(* CODESYS project CodesysV3.export

Project tree, tasks and I/O mapping:
  application HomeAutomation
    libraries: Standard, * (System); Element Collections, 3.5.14.0 (3S - Smart Software Solutions GmbH); WagoSysStandard, 1.6.1.0 (WAGO); WagoTypesAppLED, 1.5.2.0 (WAGO); WagoAppAppLED, 1.7.2.0 (WAGO); WagoAppPlcModbus, 1.1.2.5 (WAGO); Util, 3.5.14.0 (System); BASIC, 3.3.4.0 (OSCAT); BUILDING, 1.0.0.1 (OSCAT); Common Helper for development, 1.1.0.5 (Stefan Dreyer); NETWORK, 1.3.5.3 (OSCAT); MQTT, 1.2.0.6 (Stefan Dreyer); WagoTypesEvent, 1.5.2.0 (WAGO); SysSocketAsync, 3.5.17.0 (System); SysTarget, 3.5.17.0 (System); SysSocket, * (System); SM3_Shared, 4.9.0.0 (3S - Smart Software Solutions GmbH); PRO JSON, 1.0.0.15 (Pro Electric)
    task MainTask (cyclic, interval 50 ms, priority 4) calls PLC_PRG_MAIN
    task MqttCommunication (freewheeling, priority 5) calls PLC_PRG_MQTT, DMX_SEND
    task Ping (cyclic, interval 10000 ms, priority 4) calls PRG_PING_DMX
    task RS485 (cyclic, interval 200 ms, priority 15) calls PLC_PRG_RS485
    PRG's/
      program DMX_SEND [ST]
      program PLC_PRG_MAIN [SFC]: MAIN_INIT, MOVE_COVERS, PROCESS_VIRTUAL, READ_PUSHBUTTONS, WRITE_SWITCHES
      program PLC_PRG_MQTT [SFC]: MQTT_INIT, MQTT_PUBLISH, MQTT_SUBSCRIBE
      program PLC_PRG_RS485 [SFC]: RS485_INIT, RS485_RUN
      program PRG_PING_DMX [ST]
    global variables DMXVariables
    global variables MqttVariables
    global variables PersistentVars
  data type Dimmer
  data type DIMMER_CURVE
  data type VIRTUAL_MODES
  Mqtt/
    data type MQTT_MESSAGE
    function block FB_MqttPublishQueue [ST]: AddMessage, GetMessage, Reset
    function block FB_MqttPublishWorker [ST]: Init, PublishMessage
  MqttDiscovery/
    Messages/
      data type MQTT_DISCOVERY_AVTY_T
      data type MQTT_DISCOVERY_BASE
      data type MQTT_DISCOVERY_BINARY_SENSOR
      data type MQTT_DISCOVERY_BINARY_SENSOR_ENT_CAT
      data type MQTT_DISCOVERY_COVER
      data type MQTT_DISCOVERY_DEVICE
      data type MQTT_DISCOVERY_LIGHT
      data type MQTT_DISCOVERY_LIGHT_DIMMER
      data type MQTT_DISCOVERY_LOCK
      data type MQTT_DISCOVERY_SENSOR
      data type MQTT_DISCOVERY_SENSOR_ENT_CAT
      data type MQTT_DISCOVERY_SIREN
      data type MQTT_DISCOVERY_SWITCH
  RS485/
    data type RS485_EASTRON_SDM_Devices
    data type RS485_RtuQuery
    interface RS485Device: GetRtuQuery, ProcessDataArray, RequestBusTime
    function block FB_RS485_BUSCONTROLLER [ST]: Init, RegisterDevice, ReleaseBus, SetBusOccupied
  function block FB_BASE_MQTT_DISCOVERY_DEVICE [ST]: CreateBinarySensorEntity, CreateBinarySensorEntityWithCategory, CreateCoverEntity, CreateLightDimmerEntity, CreateLightEntity, CreateLockEntity, CreateSensorEntity, CreateSensorEntityWithCategory, CreateSirenEntity, CreateSwitchEntity, initBaseDevice, SendLogMessage
  function block FB_INPUT_BINARYSENSOR_MQTT [ST]: ConfigureFunctionBlock, InitMqtt, InitMqttDiscovery
  function block FB_INPUT_PUSHBUTTON_DIMMER_MQTT [ST]: ConfigureFunctionBlock, InitMqtt
  function block FB_INPUT_PUSHBUTTON_MQTT [ST]: ConfigureFunctionBlock, InitMqtt, InitMqttDiscovery
  function block FB_MQTT_BASE [ST]: InitBaseMqtt
  function block FB_MQTT_LOG [ST]: InitMqtt, InitMqttDiscovery, send
  function block FB_OUTPUT_BINARY_MQTT [ST]: InitMqtt, InitMqttDiscoveryAsLight, InitMqttDiscoveryAsLock, InitMqttDiscoveryAsSiren, InitMqttDiscoveryAsSwitch, PublishReceived
  function block FB_OUTPUT_BISTABLE_MQTT [ST]: ConfigureFunctionBlock, InitMqtt, InitMqttDiscoveryAsLight, InitMqttDiscoveryAsLock, InitMqttDiscoveryAsSiren, InitMqttDiscoveryAsSwitch, PublishReceived
  function block FB_OUTPUT_COVER_MQTT [ST]: ConfigureFunctionBlock, InitMqtt, InitMqttDiscovery, PublishReceived
  function block FB_OUTPUT_DIMMER_MQTT [ST]: ConfigureFunctionBlock, initDMX, InitMqtt, InitMqttDiscovery, PublishReceived
  function block FB_PLC_MQTT_DISCOVERY_DEVICE [ST]: GetIpAddress, GetMac, initPlcDevice
  function block FB_RS485_DUCO_DUCOBOX_MQTT [ST]: AddNode, GetRtuQuery, InitMqtt, InitRS485, ProcessDataArray, PublishReceived, PubMqttMessage, RequestBusTime
  function block FB_RS485_DUCO_DUCOBOX_NODE_MQTT [ST]: GetRtuQuery, InitMqtt, InitNode, ProcessDataArray, PubMqttMessage, RequestBusTime
  function block FB_RS485_EASTRON_SDM_POWER_MQTT [ST]: GetRtuQuery, InitMqtt, InitRS485, ProcessDataArray, PubMqttMessage, RequestBusTime
  function block FB_RS485_EASTRON_SDM220_MQTT [ST]: GetRtuQuery, InitMqtt, InitRS485, ProcessDataArray, PubMqttMessage, RequestBusTime
  function block FB_RS485_ESERA_1WIRE_GATEWAY_MQTT [ST]: EnableOwd, GetRtuQuery, InitMqtt, InitRS485, ProcessDataArray, RequestBusTime
  function block FB_RS485_ESERA_OWD_MQTT [ST]: GetRtuQuery, InitMqtt, InitOwd, ProcessAirQuality, ProcessBrigthness, ProcessDataArray, ProcessDewPoint, ProcessHumidity, ProcessOwdVoltage, ProcessTemperature, PubMqttMessage, RequestBusTime
  function block FB_VIRTUAL_BOOL_MQTT [ST]: ConfigureFunctionBlockAsVirtualInput, ConfigureFunctionBlockAsVirtualOutput, InitMqtt, PublishReceived, SetValue
  function block FB_VIRTUAL_INT_MQTT [ST]: ConfigureFunctionBlockAsVirtualInput, ConfigureFunctionBlockAsVirtualOutput, InitMqtt, PublishReceived, SetValue
  function block FB_VIRTUAL_REAL_MQTT [ST]: ConfigureFunctionBlockAsVirtualInput, ConfigureFunctionBlockAsVirtualOutput, InitMqtt, PublishReceived, SetValue
  function block FB_VIRTUAL_STRING_MQTT [ST]: ConfigureFunctionBlockAsVirtualInput, ConfigureFunctionBlockAsVirtualOutput, InitMqtt, PublishReceived, SetValue
  function SwapWordsToReal [ST]
*)

// Dimmer
{attribute 'to_string' := ''}
TYPE Dimmer :
(
	idle,
	soft_turn_on_restore,
	soft_turn_off,
	quick_turn_on,
	quick_turn_off,
	ramp_up_or_down,
	low_or_high_entering,
	low_or_high_leaving,
	low_or_high_released_by_user,
	blink
);
END_TYPE

// DIMMER_CURVE
TYPE DIMMER_CURVE :
(
	linear,
	logarithmic,
	cubic
);
END_TYPE

// VIRTUAL_MODES
TYPE VIRTUAL_MODES :
(
	Input,
	Output
);
END_TYPE

// Mqtt/MQTT_MESSAGE
TYPE MQTT_MESSAGE :
STRUCT
	Payload: STRING(1500);
	Topic: STRING(128);
	Qos: MQTT.QoS;
	MqttRetain: BOOL;
END_STRUCT
END_TYPE

// RS485/RS485_EASTRON_SDM_Devices
TYPE RS485_EASTRON_SDM_Devices :
(
	SDM120,
	SDM220,
	SDM630
);
END_TYPE

// RS485/RS485_RtuQuery
TYPE RS485_RtuQuery :
STRUCT
	DeviceId: BYTE;
	FunctionCode: BYTE;
	ReadAddress: UINT;
	ReadQuantity: UINT;
	WriteAddress: UINT;
	WriteQuantity: UINT;
	WriteData: ARRAY[0..124] OF WORD;
END_STRUCT
END_TYPE

// MqttDiscovery/Messages/MQTT_DISCOVERY_AVTY_T
TYPE MQTT_DISCOVERY_AVTY_T :
STRUCT
	topic: JSONVAR;
END_STRUCT
END_TYPE

// MqttDiscovery/Messages/MQTT_DISCOVERY_BASE
TYPE MQTT_DISCOVERY_BASE :
STRUCT
	name: JSONVAR;
	/// object_id
	obj_id: JSONVAR;
	///unique_id
	uniq_id: JSONVAR;
	/// availability
	avty: ARRAY[1..2] OF MQTT_DISCOVERY_AVTY_T;
	/// availability mode
	avty_mode: JSONVAR;
	///payload_available
	pl_avail: JSONVAR;
	/// payload_not_available
	pl_not_avail: JSONVAR;
	/// device
	dev: MQTT_DISCOVERY_DEVICE;
	/// mqtt qos
	qos: JSONVAR;
	/// extra metadata
	meta: JSONVAR;
END_STRUCT
END_TYPE

// MqttDiscovery/Messages/MQTT_DISCOVERY_BINARY_SENSOR
TYPE MQTT_DISCOVERY_BINARY_SENSOR EXTENDS MQTT_DISCOVERY_BASE :
STRUCT
	///state_topic
	stat_t: JSONVAR;
	///payload_on
	pl_on: JSONVAR;
	///payload_off
	pl_off: JSONVAR;
	/// device class
	dev_cla: JSONVAR;
END_STRUCT
END_TYPE

// MqttDiscovery/Messages/MQTT_DISCOVERY_BINARY_SENSOR_ENT_CAT
TYPE MQTT_DISCOVERY_BINARY_SENSOR_ENT_CAT EXTENDS MQTT_DISCOVERY_BINARY_SENSOR :
STRUCT
	/// entity category
	ent_cat: JSONVAR;
END_STRUCT
END_TYPE

// MqttDiscovery/Messages/MQTT_DISCOVERY_COVER
TYPE MQTT_DISCOVERY_COVER EXTENDS MQTT_DISCOVERY_BASE :
STRUCT
	///command_topic
	cmd_t: JSONVAR;
	/// payload open
	pl_open: JSONVAR;
	/// payload_close
	pl_cls: JSONVAR;
	/// payload_stop
	pl_stop: JSONVAR;
	/// state topic
	stat_t: JSONVAR;
	/// state open
	stat_open: JSONVAR;
	/// state closed	
	stat_clsd: JSONVAR;
	///  optimistic
	opt: JSONVAR;
	/// device class
	dev_cla: JSONVAR;
END_STRUCT
END_TYPE

// MqttDiscovery/Messages/MQTT_DISCOVERY_DEVICE
TYPE MQTT_DISCOVERY_DEVICE :
STRUCT
	name: JSONVAR;
	///configuration_url
	cu: JSONVAR;
	///identifiers
	ids: JSONVAR;
	///manufacturer
	mf: JSONVAR;
	///model
	mdl: JSONVAR;
	///sw_version
	sw: JSONVAR;
	///hw_version
	hw: JSONVAR;
END_STRUCT
END_TYPE

// MqttDiscovery/Messages/MQTT_DISCOVERY_LIGHT
TYPE MQTT_DISCOVERY_LIGHT EXTENDS MQTT_DISCOVERY_BASE :
STRUCT
	///command_topic
	cmd_t: JSONVAR;
	/// payload_on
	pl_on: JSONVAR;
	/// payload_off
	pl_off: JSONVAR;
	/// state_topic
	stat_t: JSONVAR;
	///  optimistic
	opt: JSONVAR;
END_STRUCT
END_TYPE

// MqttDiscovery/Messages/MQTT_DISCOVERY_LIGHT_DIMMER
TYPE MQTT_DISCOVERY_LIGHT_DIMMER EXTENDS MQTT_DISCOVERY_LIGHT :
STRUCT
	///brightness state topic
	bri_stat_t: JSONVAR;
	/// brightness command topic
	bri_cmd_t: JSONVAR;
	/// brightness scale
	bri_scl: JSONVAR;
	/// on command type
	on_cmd_type: JSONVAR;
	/// DMX
	dmxChannel: JSONVAR;
	dmxWidth: JSONVAR;
	dmxUniverse: JSONVAR;
END_STRUCT
END_TYPE

// MqttDiscovery/Messages/MQTT_DISCOVERY_LOCK
TYPE MQTT_DISCOVERY_LOCK EXTENDS MQTT_DISCOVERY_BASE :
STRUCT
	///command_topic
	cmd_t: JSONVAR;
	/// payload lock
	pl_lock: JSONVAR;
	/// payload unlock
	pl_unlk: JSONVAR;
	/// state_topic
	stat_t: JSONVAR;
	/// state locked
	stat_locked: JSONVAR;
	/// state unlocked
	stat_unlocked: JSONVAR;
	///  optimistic
	opt: JSONVAR;
END_STRUCT
END_TYPE

// MqttDiscovery/Messages/MQTT_DISCOVERY_SENSOR
TYPE MQTT_DISCOVERY_SENSOR EXTENDS MQTT_DISCOVERY_BASE :
STRUCT
	///state_topic
	stat_t: JSONVAR;
	///expire after
	exp_aft: JSONVAR;
END_STRUCT
END_TYPE

// MqttDiscovery/Messages/MQTT_DISCOVERY_SENSOR_ENT_CAT
TYPE MQTT_DISCOVERY_SENSOR_ENT_CAT EXTENDS MQTT_DISCOVERY_SENSOR :
STRUCT
	/// entity category
	ent_cat: JSONVAR;
END_STRUCT
END_TYPE

// MqttDiscovery/Messages/MQTT_DISCOVERY_SIREN
TYPE MQTT_DISCOVERY_SIREN EXTENDS MQTT_DISCOVERY_BASE :
STRUCT
	///command_topic
	cmd_t: JSONVAR;
	/// payload_on
	pl_on: JSONVAR;
	/// payload_off
	pl_off: JSONVAR;
	/// state_topic
	stat_t: JSONVAR;
	/// state on
	stat_on: JSONVAR;
	/// state off
	stat_off: JSONVAR;
	///  optimistic
	opt: JSONVAR;
END_STRUCT
END_TYPE

// MqttDiscovery/Messages/MQTT_DISCOVERY_SWITCH
TYPE MQTT_DISCOVERY_SWITCH EXTENDS MQTT_DISCOVERY_BASE :
STRUCT
	///command_topic
	cmd_t: JSONVAR;
	/// payload_on
	pl_on: JSONVAR;
	/// payload_off
	pl_off: JSONVAR;
	/// state_topic
	stat_t: JSONVAR;
	/// state on
	stat_on: JSONVAR;
	/// state off
	stat_off: JSONVAR;
	///  optimistic
	opt: JSONVAR;
	/// device class
	dev_cla: JSONVAR;
END_STRUCT
END_TYPE

// HomeAutomation/DMXVariables
{attribute 'qualified_only'}
VAR_GLOBAL
	// unicast: 10.1.1.4
	// multicast: 10.1.1.255  
	// broadcast: 255.255.255.255  
	IP						: STRING:='10.1.1.4'; 
	DMX 					: oscat_network.NETWORK_BUFFER_SHORT;
END_VAR

// HomeAutomation/MqttVariables
{attribute 'qualified_only'}
VAR_GLOBAL	
	(* Broker setup *)
	clientID				:STRING:='PLC-House';
	broker					:STRING:='192.168.1.52:1883'; 	
	(* use the below for username password authentication to broker *)
	(* broker					:STRING:='user:password@192.168.1.36:1883'; *)
	

	(* Shared Variables for MQTT publish communication *)
	fbMqttPublishQueue		:FB_MqttPublishQueue;  
	
	(* Shared Variables for MQTT subscribe communication *)	
	collector_FB_OUTPUT_SWITCH_MQTT		:MQTT.CallbackCollector;		
	collector_FB_OUTPUT_COVER_MQTT		:MQTT.CallbackCollector;	
	collector_FB_VIRTUAL_MQTT			:MQTT.CallbackCollector;		
	collector_FB_DIMMER_MQTT			:MQTT.CallbackCollector;
	collector_FB_MQTT_LOG				:MQTT.CallbackCollector;	
	collector_FB_RS485_MQTT				:MQTT.CallbackCollector;
	
	(* QOS Constants *)
	MQTT_QOS_EXACTLY_ONCE				:MQTT.QoS := MQTT.QoS.ExactlyOnce;
	 
	
	(* HOME ASSISTANT DISCOVERY VIA MQTT*)
	PLC_Device						:FB_PLC_MQTT_DISCOVERY_DEVICE;	
	
	(* Topics *)
	MqttMain						:STRING(16) := 'Devices/';
	MqttType						:STRING(16) := 'PLC/';
	MqttDevice						:STRING(16) := 'House/';
	// e.g. Devices/PLC/House
	MqttBaseTopic					:STRING(100) := CONCAT(CONCAT(MqttMain,MqttType),MqttDevice);
	MqttDiagnosticTopic				:STRING(100) := CONCAT(MqttBaseTopic,'diagnostic');									
	MqttAvailabilityTopic 			:STRING(100) := CONCAT(MqttBaseTopic,'availability');							
	MqttAvailabilityOnlinePayload	:STRING(20) := 'online';							
	MqttAvailabilityOfflinePayload	:STRING(20) := 'offline';
	MQTTAvailabilityHartbeatTime	:TIME:=T#5S;
	MqttHADiscoveryPrefix			:STRING(16) := 'homeassistant/';
	
	(* FB Topics *)
	MqttPushbuttonPrefix			:STRING(100) := CONCAT(MqttBaseTopic,'Out/DigitalInputs/Pushbuttons/');
	MqttPubSwitchPrefix				:STRING(100) := CONCAT(MqttBaseTopic,'Out/DigitalOutputs/');
	MqttSubSwitchPrefix				:STRING(100) := CONCAT(MqttBaseTopic,'In/DigitalOutputs/');
	MqttPubCoverPrefix				:STRING(100) := CONCAT(MqttBaseTopic,'Out/Covers/');
	MqttSubCoverPrefix				:STRING(100) := CONCAT(MqttBaseTopic,'In/Covers/');
	MqttPubDimmerPrefix				:STRING(100) := CONCAT(MqttBaseTopic,'Out/Dimmers/');
	MqttSubDimmerPrefix				:STRING(100) := CONCAT(MqttBaseTopic,'In/Dimmers/');
	MqttPubVirtualPrefix			:STRING(100) := CONCAT(MqttBaseTopic,'Out/Virtuals/');
	MqttSubVirtualPrefix			:STRING(100) := CONCAT(MqttBaseTopic,'In/Virtuals/');
	MqttPubRS485Prefix				:STRING(100) := CONCAT(MqttBaseTopic,'Out/RS485/');
	MqttSubRS485Prefix				:STRING(100) := CONCAT(MqttBaseTopic,'In/RS485/');
	
	(* Wildcard subscriptions *)
	MqttSubSwitchTopic				:STRING(100) := CONCAT(MqttSubSwitchPrefix,'+');
	MqttSubCoverTopic				:STRING(100) := CONCAT(MqttSubCoverPrefix,'+');
	MqttSubVirtualTopic				:STRING(100) := CONCAT(MqttSubVirtualPrefix,'+');
	MqttSubDimmerTopic				:STRING(100) := CONCAT(MqttSubDimmerPrefix,'#');
	MqttSubRS485Topic				:STRING(100) := CONCAT(MqttSubRS485Prefix,'#');

END_VAR

// HomeAutomation/PersistentVars
{attribute 'qualified_only'}
VAR_GLOBAL PERSISTENT RETAIN
	// Generated instance path of persistent variable
	PLC_PRG_MAIN.FB_DO_BIN_001.PreviousState: BOOL;
	// Generated instance path of persistent variable
	PLC_PRG_MAIN.FB_DO_COVER_001.internalDir: BOOL;
	// Generated instance path of persistent variable
	PLC_PRG_MAIN.FB_AO_DIMMER_001.PreviousOUT: BYTE;
	// Generated instance path of persistent variable
	PLC_PRG_MAIN.FB_AO_DIMMER_001.PreviousQ: BOOL;
	// Generated instance path of persistent variable
	PLC_PRG_MAIN.FB_VIRTUAL_INT_001.PreviousState: INT;
	// Generated instance path of persistent variable
	PLC_PRG_MAIN.FB_VIRTUAL_BOOL_001.PreviousState: BOOL;
	// Generated instance path of persistent variable
	PLC_PRG_MAIN.FB_VIRTUAL_STRING_001.PreviousState: STRING;
	// Generated instance path of persistent variable
	PLC_PRG_MAIN.FB_VIRTUAL_REAL_001.PreviousState: REAL;
END_VAR

// HomeAutomation/PRG's/PLC_PRG_MAIN
PROGRAM PLC_PRG_MAIN
VAR		
	(* INPUT FUNCTION BLOCKS *)
	FB_DI_PB_001				:FB_INPUT_PUSHBUTTON_MQTT;
	FB_DI_PB_002				:FB_INPUT_PUSHBUTTON_DIMMER_MQTT;
	
	(* OUTPUT FUNCTION BLOCKS *)
	FB_DO_BIN_001				:FB_OUTPUT_BINARY_MQTT;
	FB_DO_BISTABLE_001			:FB_OUTPUT_BISTABLE_MQTT;

	(* COVER FUNCTION BLOCKS *)
	FB_DO_COVER_001				:FB_OUTPUT_COVER_MQTT;
	
	(* DIMMER FUNCTION BLOCKS *)
	FB_AO_DIMMER_001			:FB_OUTPUT_DIMMER_MQTT;	
	TestOUT						:WORD;
	
	(* VIRTUAL FUNCTION BLOCKS *)
	FB_VIRTUAL_INT_001				:FB_VIRTUAL_INT_MQTT;
	FB_VIRTUAL_BOOL_001				:FB_VIRTUAL_BOOL_MQTT;
	FB_VIRTUAL_STRING_001			:FB_VIRTUAL_STRING_MQTT;
	FB_VIRTUAL_REAL_001				:FB_VIRTUAL_REAL_MQTT;
END_VAR

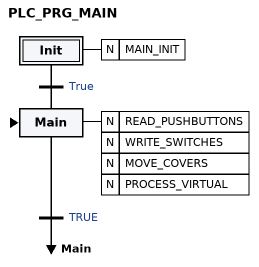
INITIAL_STEP Init:
    MAIN_INIT(N);
END_STEP
TRANSITION FROM Init TO Main
    := True;
END_TRANSITION
STEP Main:
    READ_PUSHBUTTONS(N);
    WRITE_SWITCHES(N);
    MOVE_COVERS(N);
    PROCESS_VIRTUAL(N);
END_STEP
TRANSITION FROM Main TO Main
    := TRUE;
END_TRANSITION

ACTION MAIN_INIT:
(* MQTT Discovery device*)
MqttVariables.PLC_Device.initPlcDevice(
	MqttDiscoveryPrefix := MqttVariables.MqttHADiscoveryPrefix,
	pMqttPublishQueue := ADR(MqttVariables.fbMqttPublishQueue),
	availabilityTopic := MqttVariables.MqttAvailabilityTopic,
	availabilityOnline := MqttVariables.MqttAvailabilityOnlinePayload,
	availabilityOffline := MqttVariables.MqttAvailabilityOfflinePayload,
	MqttDiagnosticTopic := MqttVariables.MqttDiagnosticTopic
);


(* INIT DIGITAL INPUT STUFF *)
FB_DI_PB_001.InitMqtt(
	MQTTPublishPrefix:= ADR(MqttVariables.MqttPushbuttonPrefix),	(* pointer to string prefix for the mqtt publish topic *)
	pMqttPublishQueue := ADR(MqttVariables.fbMqttPublishQueue)		(* pointer to MqttPublishQueue to send a new Mqtt event *)
);

FB_DI_PB_001.InitMqttDiscovery(
	name := 'Button number 001',						(* The name show in Home Assistant frond-end*)
	Device := ADR(MqttVariables.PLC_Device),							(* The device show in Home Assistant *)
);

FB_DI_PB_002.InitMqtt(
	MQTTPublishPrefix:= ADR(MqttVariables.MqttPushbuttonPrefix),	
	pMqttPublishQueue := ADR(MqttVariables.fbMqttPublishQueue),
    TRUE,                                                               (* specify whether dimmer value should be outputted on MQTT topic *)
    MQTT.QoS.ExactlyOnce,                                            (* specify the QoS for the dimmer mqtt events (values 0-255) *)    
    5                                                                   (* specify the resolution for the dimmer mqtt events *)    
);


(* ALTER THE DIMMER OUTPUT DEFAULT BEHAVIOR *)
FB_AO_DIMMER_001.ConfigureFunctionBlock(
	T_Debounce:=T#10MS,
	T_Reconfig:=T#10S,
	T_On_Max:=T#0S,
	T_Dimm_Start:=T#400MS,
	T_Dimm:=T#3S,
	Min_On:=50,
	Max_On:=255,
	Soft_Dimm:=TRUE,
	Rst_Out:=FALSE,
	OUT_LinearScaleMin:=11000,
	OUT_LinearScaleMax:=32767
);

(* INIT DMX / ART-NET OUTPUT, OPTIONAL*)
FB_AO_DIMMER_001.InitDmx(
	DmxChannel := 1,							(* The channel *)
	DmxWidth:=1, 								(* Width of DMX channel, 1 or 2, aka 8 or 16 bit *)
	pDmxValues := ADR(DMXVariables.DMX.BUFFER), (* pointer to network buffer *)
	DmxUniverse:=1								(* Universe, but the buffer desides, this is only meta data that ends up in MQTT*)
);

(* INIT HOME ASSISTANT DISCOVERTY*)
FB_AO_DIMMER_001.InitMqttDiscovery(
	name := '001. Office strip cold',					(* The name show in Home Assistant frond-end*)
	Device := ADR(MqttVariables.PLC_Device),							(* The device show in Home Assistant *)
);


(* INIT DIGITAL OUTPUT STUFF *)
FB_DO_BISTABLE_001.InitMqtt(
	MQTTPublishPrefix:= ADR(MqttVariables.MqttPubSwitchPrefix),					(* pointer to string prefix for the mqtt publish topic *)
	MQTTSubscribePrefix:= ADR(MqttVariables.MqttSubSwitchPrefix),				(* pointer to string prefix for the mqtt subscribe topic *)
	pMqttPublishQueue := ADR(MqttVariables.fbMqttPublishQueue),					(* pointer to MqttPublishQueue to send a new Mqtt event *)
	pMqttCallbackCollector := ADR(MqttVariables.collector_FB_OUTPUT_SWITCH_MQTT)(* pointer to CallbackCollector to receive Mqtt subscription events *)
);

FB_DO_BISTABLE_001.InitMqttDiscoveryAsLight(
	name := 'light number 1',						(* The name show in Home Assistant frond-end*)
	Device := ADR(MqttVariables.PLC_Device),							(* The device show in Home Assistant *)
);

FB_DO_BIN_001.InitMqtt(
	MQTTPublishPrefix:= ADR(MqttVariables.MqttPubSwitchPrefix),					(* pointer to string prefix for the mqtt publish topic *)
	MQTTSubscribePrefix:= ADR(MqttVariables.MqttSubSwitchPrefix),				(* pointer to string prefix for the mqtt subscribe topic *)
	pMqttPublishQueue := ADR(MqttVariables.fbMqttPublishQueue),					(* pointer to MqttPublishQueue to send a new Mqtt event *)
	pMqttCallbackCollector := ADR(MqttVariables.collector_FB_OUTPUT_SWITCH_MQTT)(* pointer to CallbackCollector to receive Mqtt subscription events *)
);

FB_DO_BIN_001.InitMqttDiscoveryAsLight(
	name := 'light number 2',						(* The name show in Home Assistant frond-end*)
	Device := ADR(MqttVariables.PLC_Device),							(* The device show in Home Assistant *)
);

(* INIT COVERS STUFF *)
FB_DO_COVER_001.InitMqtt(MQTTPublishPrefix:= ADR(MqttVariables.MqttPubCoverPrefix),	(* pointer to string prefix for the mqtt publish topic *)
	MQTTSubscribePrefix:= ADR(MqttVariables.MqttSubCoverPrefix),					(* pointer to string prefix for the mqtt subscribe topic *)
	pMqttPublishQueue := ADR(MqttVariables.fbMqttPublishQueue),						(* pointer to MqttPublishQueue to send a new Mqtt event *)
	pMqttCallbackCollector := ADR(MqttVariables.collector_FB_OUTPUT_COVER_MQTT)  	(* pointer to CallbackCollector to receive Mqtt subscription events *)
);

FB_DO_COVER_001.initmqttdiscovery(								(*see dimmer for full example *)
	name := 'cover number 001',									(* the name show in home assistant frond-end*)
	device := ADR(MqttVariables.PLC_Device),										(* the device show in home assistant *)
);

FB_DO_COVER_001.ConfigureFunctionBlock(
	T_LOCKOUT:=T#1S,											(* delay between change of direction *)
	T_UD:=T#20S													(* run time to move the cover completely up/down *)
);


(* INIT VIRTUAL STUFF *)
FB_VIRTUAL_STRING_001.InitMqtt(MQTTPublishPrefix:= ADR(MqttVariables.MqttPubVirtualPrefix),				
	MQTTSubscribePrefix:= ADR(MqttVariables.MqttSubVirtualPrefix),									
	pMqttPublishQueue := ADR(MqttVariables.fbMqttPublishQueue),						
	pMqttCallbackCollector := ADR(MqttVariables.collector_FB_VIRTUAL_MQTT),
	MqttQos:=MQTT.QoS.ExactlyOnce, 
	MqttRetain:=FALSE									
);
FB_VIRTUAL_STRING_001.ConfigureFunctionBlockAsVirtualInput(DefaultValue:='HelloWorld',SetDefaultValueStartup:=TRUE,PublishAtStartup:=TRUE,UsePersistentAtStartup:=FALSE,ConfirmReceival:=TRUE);


FB_VIRTUAL_INT_001.InitMqtt(MQTTPublishPrefix:= ADR(MqttVariables.MqttPubVirtualPrefix),				
	MQTTSubscribePrefix:= ADR(MqttVariables.MqttSubVirtualPrefix),									
	pMqttPublishQueue := ADR(MqttVariables.fbMqttPublishQueue),						
	pMqttCallbackCollector := ADR(MqttVariables.collector_FB_VIRTUAL_MQTT),
	MqttQos:=MQTT.QoS.ExactlyOnce, 
	MqttRetain:=FALSE												
);
FB_VIRTUAL_INT_001.ConfigureFunctionBlockAsVirtualInput(DefaultValue:=0,SetDefaultValueStartup:=TRUE,PublishAtStartup:=TRUE,UsePersistentAtStartup:=FALSE,ConfirmReceival:=TRUE);
(* FB_VIRTUAL_INT_001.ConfigureFunctionBlockAsVirtualOutput(PublishAtStartup:=TRUE); *)


FB_VIRTUAL_BOOL_001.InitMqtt(MQTTPublishPrefix:= ADR(MqttVariables.MqttPubVirtualPrefix),				
	MQTTSubscribePrefix:= ADR(MqttVariables.MqttSubVirtualPrefix),									
	pMqttPublishQueue := ADR(MqttVariables.fbMqttPublishQueue),						
	pMqttCallbackCollector := ADR(MqttVariables.collector_FB_VIRTUAL_MQTT),
	MqttQos:=MQTT.QoS.ExactlyOnce, 
	MqttRetain:=FALSE											
);
(* FB_VIRTUAL_BOOL_001.ConfigureFunctionBlockAsVirtualInput(DefaultValue:=FALSE,SetDefaultValueStartup:=TRUE,PublishAtStartup:=TRUE,UsePersistentAtStartup:=FALSE); *)
FB_VIRTUAL_BOOL_001.ConfigureFunctionBlockAsVirtualOutput(PublishAtStartup:=TRUE);

FB_VIRTUAL_REAL_001.InitMqtt(MQTTPublishPrefix:= ADR(MqttVariables.MqttPubVirtualPrefix),				
	MQTTSubscribePrefix:= ADR(MqttVariables.MqttSubVirtualPrefix),									
	pMqttPublishQueue := ADR(MqttVariables.fbMqttPublishQueue),						
	pMqttCallbackCollector := ADR(MqttVariables.collector_FB_VIRTUAL_MQTT),
	MqttQos:=MQTT.QoS.ExactlyOnce, 
	MqttRetain:=FALSE												
);
FB_VIRTUAL_REAL_001.ConfigureFunctionBlockAsVirtualInput(DefaultValue:=0.1,SetDefaultValueStartup:=TRUE,PublishAtStartup:=TRUE,UsePersistentAtStartup:=FALSE,ConfirmReceival:=TRUE);
(* FB_VIRTUAL_REAL_001.ConfigureFunctionBlockAsVirtualOutput(PublishAtStartup:=TRUE); *)



MqttVariables.PLC_Device.SendLogMessage('Init finished', 'MAIN_INIT');
END_ACTION

ACTION MOVE_COVERS:
FB_DO_COVER_001(
	TOGGLE:=FB_DI_PB_001.P_LONG,
	MU=>DO_031,
	MD=>DO_032	
);
END_ACTION

ACTION PROCESS_VIRTUAL:

FB_VIRTUAL_BOOL_001();
FB_VIRTUAL_INT_001();
FB_VIRTUAL_STRING_001();
FB_VIRTUAL_REAL_001();
END_ACTION

ACTION READ_PUSHBUTTONS:
FB_DI_PB_001(PB:= DI_001); (* Provide the input FB the correct phyical input to validate each cyclus *)
FB_DI_PB_002(PB:= DI_002);
END_ACTION

ACTION WRITE_SWITCHES:
FB_DO_BIN_001(OUT	=>		DO_001,										(* couple the function block to the physical output *)
	PRIO_HIGH				:=FALSE,  									(* brings the output high regardless of other input values *)
	PRIO_LOW				:=FALSE, 									(* brings the output low regardless of other input values. NOTE: PRIO_HIGH overrules PRIO_LOW input *)
	TOGGLE					:=FB_DI_PB_001.SINGLE 						(* for toggling the output *)	
);

FB_AO_DIMMER_001(
	SINGLE:=FB_DI_PB_001.SINGLE,
	LONG:=FB_DI_PB_001.LONG, 
	P_LONG:=FB_DI_PB_001.P_LONG, 
	Q_OUT => TestOUT,
	SET:=  FB_DI_PB_001.DOUBLE,
	VAL:=125
);

FB_DO_BISTABLE_001();
END_ACTION

END_PROGRAM

// FB_INPUT_PUSHBUTTON_MQTT
{attribute 'reflection' := ''}
FUNCTION_BLOCK FB_INPUT_PUSHBUTTON_MQTT EXTENDS FB_MQTT_BASE
VAR_INPUT
	PB: BOOL;
END_VAR
VAR_OUTPUT
	SINGLE: BOOL;
	DOUBLE: BOOL;
	LONG: BOOL;
	P_LONG: BOOL;
END_VAR
VAR
	/// Refelection: object's full instance name
	{attribute 'instance-path' := ''}
	{attribute 'noinit'}
	InstancePath: STRING;
	FB_DETECTPUSH: OSCAT_BUILDING.CLICK_MODE;
	P_LONG_R_TRIG: Standard.R_TRIG;
	P_LONG_F_TRIG: Standard.F_TRIG;
	/// Default value for click mode, can be overwritten by method call 
	T_Long: TIME := TIME#400ms;
	MqttDiscoveryMessage: MQTT_DISCOVERY_SENSOR;
END_VAR

FB_DETECTPUSH(
	IN:= PB, 	
	SINGLE=> SINGLE, 
	DOUBLE=> DOUBLE, 
	TP_LONG=> LONG, 
	LONG=> P_LONG,
	T_LONG:= T_Long);
	
P_LONG_R_TRIG(CLK:=FB_DETECTPUSH.LONG);
P_LONG_F_TRIG(CLK:=FB_DETECTPUSH.LONG);
	
IF FB_DETECTPUSH.SINGLE AND InitMqttDone THEN
	pMqttPublishQueue^.AddMessage(
		Payload := 'SINGLE',
		Topic := CONCAT(MqttPublishTopicPrefix^, MqttPublishTopicSuffix),
		Qos := MQTT.QoS.ExactlyOnce,
		MqttRetain := FALSE
	);
END_IF

IF FB_DETECTPUSH.DOUBLE AND InitMqttDone THEN
	pMqttPublishQueue^.AddMessage(
		Payload := 'DOUBLE',
		Topic := CONCAT(MqttPublishTopicPrefix^, MqttPublishTopicSuffix),
		Qos := MQTT.QoS.ExactlyOnce,
		MqttRetain := FALSE
	);
END_IF

IF FB_DETECTPUSH.TP_LONG AND InitMqttDone THEN
	pMqttPublishQueue^.AddMessage(
		Payload := 'LONG',
		Topic := MQTTPublishTopic,
		Qos := MQTT.QoS.ExactlyOnce,
		MqttRetain := FALSE
	);
END_IF

IF P_LONG_F_TRIG.Q AND InitMqttDone THEN
	pMqttPublishQueue^.AddMessage(
		Payload := 'RELEASED',
		Topic := MQTTPublishTopic,
		Qos := MQTT.QoS.ExactlyOnce,
		MqttRetain := FALSE
	);
END_IF



IF (P_LONG_R_TRIG.Q OR P_LONG_F_TRIG.Q) AND InitMqttDone THEN
	

	pMqttPublishQueue^.AddMessage(
		Payload := BOOL_TO_STRING(FB_DETECTPUSH.LONG),
		Topic := CONCAT(MQTTPublishTopic,'/P_LONG'),
		Qos := MQTT.QoS.ExactlyOnce,
		MqttRetain := TRUE
	);
END_IF

METHOD ConfigureFunctionBlock
VAR_INPUT
	/// Default value for click mode, can be overwritten by method call 
	T_Long: TIME;
END_VAR
THIS^.T_Long:=T_Long;
END_METHOD

METHOD InitMqtt
VAR_INPUT
	MQTTPublishPrefix: POINTER TO STRING;
	pMqttPublishQueue: POINTER TO FB_MqttPublishQueue;
END_VAR
SUPER^._InstancePath := THIS^.InstancePath; // Due to reflection its location is important

(*pass trough*)
THIS^.pMqttPublishQueue := pMqttPublishQueue;
THIS^.MqttPublishTopicPrefix:=MQTTPublishPrefix;
SUPER^.InitBaseMqtt();
END_METHOD

METHOD InitMqttDiscovery
VAR_INPUT
	Device: POINTER TO FB_PLC_MQTT_DISCOVERY_DEVICE;
	Name: STRING(255);
	overruleId: STRING(255) := '';
	meta: STRING(255) := '';
END_VAR
VAR
	id: STRING(255);
END_VAR
IF InitMqttDone AND NOT initMqttDiscoveryDone THEN
	
	IF CommonTypesAndFunctions.StrEquals(str1:= ADR(overruleId), str2:= ADR('')) THEN
		id := CONCAT(CONCAT(THIS^.DeviceName,'_'), THIS^.InstanceNamePt^); // 'FB_DI_PB_003'
	ELSE
		id := overruleId; // 'MY_PH_GND_HALL_01'
	END_IF
	
	Device^.CreateSensorEntity(
		Name := name,
		Id := id,
		Meta := meta,
		StateTopic := THIS^.MQTTPublishTopic,
		ExpiryAfter := 2);

	initMqttDiscoveryDone := TRUE;
END_IF
END_METHOD

END_FUNCTION_BLOCK

// FB_MQTT_BASE
FUNCTION_BLOCK FB_MQTT_BASE
VAR
	_InstancePath: STRING;
	InstanceNamePt: POINTER TO STRING;
	DeviceName: STRING;
	InitMqttDone: BOOL;
	/// Publish (Out);
	MqttPublishTopicPrefix: POINTER TO STRING;
	MqttPublishTopicSuffix: STRING(50);
	MQTTPublishTopic: STRING(100);
	/// Subscribe (In)
	MqttSubscribeTopicPrefix: POINTER TO STRING;
	MqttSubscribeTopicSuffix: STRING(50);
	MQTTSubscribeTopic: STRING(100);
	pMqttPublishQueue: POINTER TO FB_MqttPublishQueue;
	MqttHighRequest: BOOL;
	MqttLowRequest: BOOL;
	MqttQos: MQTT.QoS := MQTT.QoS.ExactlyOnce;
	MqttRetain: BOOL := TRUE;
	/// HA Discovery specific 
	ComposeJSON: STRUCT_TO_JSON;
	initMqttDiscoveryDone: BOOL := FALSE;
END_VAR

METHOD InitBaseMqtt
VAR
	MQTTPublishPrefix: POINTER TO STRING;
	MQTTSubscribePrefix: POINTER TO STRING;
	pMqttPublishQueue: POINTER TO FB_MqttPublishQueue;
END_VAR

(*Define instance names*)
InstanceNamePt := CommonTypesAndFunctions.FindLastDot(ADR(_InstancePath)) + 1;

DeviceName := LEFT(_InstancePath,find(_InstancePath, '.' )-1  ) ;

// Publish (Out);
IF	NOT CommonTypesAndFunctions.StrEquals(ADR(MqttPublishTopicPrefix),ADR('')) THEN
	THIS^.MqttPublishTopicSuffix := InstanceNamePt^;
	THIS^.MQTTPublishTopic := CONCAT(MqttPublishTopicPrefix^, THIS^.MqttPublishTopicSuffix);
END_IF

// Subscribe (In)
IF	NOT CommonTypesAndFunctions.StrEquals(ADR(MqttSubscribeTopicPrefix),ADR('')) THEN
	THIS^.MQTTSubscribeTopicSuffix := InstanceNamePt^;
	THIS^.MQTTSubscribeTopic := CONCAT(MqttSubscribeTopicPrefix^ ,THIS^.MQTTSubscribeTopicSuffix);
END_IF

InitMqttDone := TRUE;
END_METHOD

END_FUNCTION_BLOCK

// Mqtt/FB_MqttPublishQueue
FUNCTION_BLOCK FB_MqttPublishQueue
VAR_OUTPUT
	EMPTY: BOOL := TRUE;
	FULL: BOOL;
END_VAR
VAR
	localMessage: MQTT_MESSAGE;
	fifo: ARRAY[0..n] OF MQTT_MESSAGE;
	pr: INT;
	pw: INT;
END_VAR
VAR CONSTANT
	/// changing this value will chage the number of stored elements in the fifo 
	n: INT := 1024;
END_VAR

METHOD AddMessage
VAR_INPUT
	Payload: STRING(1500);
	Topic: STRING(128);
	Qos: MQTT.QoS;
	MqttRetain: BOOL;
END_VAR
IF NOT FULL THEN
	localMessage.Payload := Payload;
	localMessage.Topic := Topic;
	localMessage.Qos := Qos;
	localMessage.MqttRetain := MqttRetain;
	fifo[pw] := localMessage;
	pw := OSCAT_BASIC.INC1(pw,n);
	FULL := pw = pr;
	EMPTY := FALSE;
END_IF;
END_METHOD

METHOD GetMessage : MQTT_MESSAGE
IF NOT EMPTY THEN
	GetMessage := fifo[pr];
	pr := OSCAT_BASIC.INC1(pr,n);
	EMPTY := pr = pw;
	FULL := FALSE;
END_IF;
END_METHOD

METHOD Reset
pw := pr;
FULL := FALSE;
EMPTY := TRUE;
END_METHOD

END_FUNCTION_BLOCK

// FB_PLC_MQTT_DISCOVERY_DEVICE
{attribute 'reflection' := ''}
FUNCTION_BLOCK FB_PLC_MQTT_DISCOVERY_DEVICE EXTENDS FB_BASE_MQTT_DISCOVERY_DEVICE
VAR
	MqttDiagnosticTopicIP: STRING;
	MqttRefreshIP: OSCAT_BASIC.GEN_PULSE;
END_VAR

(* allow the pulse generator to generate a pulse, used for refreshing IP address *)
MqttRefreshIP();

(* Refresh the IP address on every pulse *)
IF NOT(xInit) AND MqttRefreshIP.Q THEN		
	pMqttPublishQueue^.AddMessage(
		Payload:= GetIpAddress(),
		Topic := MqttDiagnosticTopicIP,
		Qos := MQTT.QoS.ExactlyOnce,
		MqttRetain := TRUE,
	);
END_IF

METHOD PRIVATE GetIpAddress : STRING(15)
VAR
	AdapterInfo: SOCK_ADAPTER_INFORMATION;
	hAdapter: RTS_IEC_HANDLE;
	udiStructSize: UDINT := SIZEOF(AdapterInfo);
	rResult: RTS_IEC_RESULT;
	xFirstAdapter: BOOL;
END_VAR
xFirstAdapter := TRUE;
rResult := 0;
WHILE rResult = 0 DO   
	IF xFirstAdapter THEN
		hAdapter := SysSockGetFirstAdapterInfo(ADR(AdapterInfo), ADR(udiStructSize), ADR(rResult));
	ELSE   
		hAdapter := SysSockGetNextAdapterInfo(hAdapter, ADR(AdapterInfo), ADR(udiStructSize), ADR(rResult));
	END_IF
	IF rResult = 0 THEN
		GetIpAddress := Standard.CONCAT(BYTE_TO_STRING(AdapterInfo.IpAddr.S_un_b.s_b1),'.');
		GetIpAddress := Standard.CONCAT(GetIpAddress,BYTE_TO_STRING(AdapterInfo.IpAddr.S_un_b.s_b2));
		GetIpAddress := Standard.CONCAT(GetIpAddress,'.');
		GetIpAddress := Standard.CONCAT(GetIpAddress,BYTE_TO_STRING(AdapterInfo.IpAddr.S_un_b.s_b3));
		GetIpAddress := Standard.CONCAT(GetIpAddress,'.');
		GetIpAddress := Standard.CONCAT(GetIpAddress,BYTE_TO_STRING(AdapterInfo.IpAddr.S_un_b.s_b4));
	END_IF
	xFirstAdapter := FALSE;   
END_WHILE
END_METHOD

METHOD PRIVATE GetMac : STRING(17)
VAR
	AdapterInfo: SOCK_ADAPTER_INFORMATION;
	hAdapter: RTS_IEC_HANDLE;
	udiStructSize: UDINT := SIZEOF(AdapterInfo);
	rResult: RTS_IEC_RESULT;
	xFirstAdapter: BOOL;
END_VAR
xFirstAdapter := TRUE;
rResult := 0;
WHILE rResult = 0 DO   
	IF xFirstAdapter THEN
		hAdapter := SysSockGetFirstAdapterInfo(ADR(AdapterInfo), ADR(udiStructSize), ADR(rResult));
	ELSE   
		hAdapter := SysSockGetNextAdapterInfo(hAdapter, ADR(AdapterInfo), ADR(udiStructSize), ADR(rResult));
	END_IF
	IF rResult = 0 THEN
		GetMac := Standard.CONCAT(SM0.Byte_To_HexString(AdapterInfo.abyMac[0]),'-');
		GetMac := Standard.CONCAT(GetMac,SM0.Byte_To_HexString(AdapterInfo.abyMac[1]));
		GetMac := Standard.CONCAT(GetMac,'-');
		GetMac := Standard.CONCAT(GetMac,SM0.Byte_To_HexString(AdapterInfo.abyMac[2]));
		GetMac := Standard.CONCAT(GetMac,'-');
		GetMac := Standard.CONCAT(GetMac,SM0.Byte_To_HexString(AdapterInfo.abyMac[3]));
		GetMac := Standard.CONCAT(GetMac,'-');
		GetMac := Standard.CONCAT(GetMac,SM0.Byte_To_HexString(AdapterInfo.abyMac[4]));
		GetMac := Standard.CONCAT(GetMac,'-');
		GetMac := Standard.CONCAT(GetMac,SM0.Byte_To_HexString(AdapterInfo.abyMac[5]));
	END_IF
	xFirstAdapter := FALSE;   
END_WHILE
END_METHOD

METHOD initPlcDevice
VAR_INPUT
	url: STRING := '';
	availabilityTopic: STRING;
	availabilityOnline: STRING;
	availabilityOffline: STRING;
	MqttDiscoveryPrefix: STRING;
	MqttDiagnosticTopic: STRING;
	pMqttPublishQueue: POINTER TO FB_MqttPublishQueue;
END_VAR
VAR
	LocalUrl: STRING;
	iSplitLocation: INT;
	iecResult: SysTypes.RTS_IEC_RESULT;
	/// must identic to the name in the device tree
	sAppName: STRING;
	pApp: POINTER TO CmpApp.APPLICATION;
	stAppInfo: CmpApp.APPLICATION_INFO;
	pstAppInfo: POINTER TO CmpApp.APPLICATION_INFO := ADR(stAppInfo);
	sIpAddr: STRING(15);
	sMacAddr: STRING(17);
	manufacturer: WSTRING;
	manufacturerSize: UDINT := SIZEOF(manufacturer);
	model: WSTRING;
	modelSize: DINT := SIZEOF(model);
	sSerialNumber: STRING;
	psSerialNumber: POINTER TO STRING := ADR(sSerialNumber);
	diSerialNumber: DINT := SIZEOF(sSerialNumber);
	CompilerVersion: Version;
	SCompilerVersion: STRING;
END_VAR
IF xInit THEN
    xInit := FALSE;
	
	(* get the appname first *)
	sAppName := PRO_JSON.GPL_JSON.ApplicationName;
	
	(* IP address and MAC *)
	sIpAddr := GetIpAddress();
	sMacAddr := GetMac();

	(* manufacturer *)
	iecResult := SysTarget.SysTargetGetVendorName(pwszName := ADR(manufacturer), pnMaxLength := ADR(manufacturerSize));
	(* model *)
    iecResult := SysTarget.SysTargetGetDeviceName(pwszName := ADR(model), pnMaxLength := ADR(modelSize));
    (* serial number *)
    iecResult := SysTarget.SysTargetGetSerialNumber(ppsSerialNumber := ADR(psSerialNumber), pnMaxLen := ADR(diSerialNumber));

	(* device name *)	
    pApp := AppFindApplicationByName(pszString := sAppName, pResult := ADR(iecResult));   
    pstAppInfo := AppGetApplicationInfo(pApp := pApp, pResult := ADR(iecResult)); 		
	iSplitLocation := COL.Stu.StrFindA(
		pst1:= ADR(THIS^.InstanceName), 
		pst2:= ADR('.'), 
		uiSearchStart:= 1
	) - 1;	
	
	(* sw version *)
	CompilerVersion := __SYSTEM.Constants.CompilerVersion;
	SCompilerVersion := CONCAT(UINT_TO_STRING(CompilerVersion.uiMajor), '.');
	SCompilerVersion := CONCAT(SCompilerVersion, UINT_TO_STRING(CompilerVersion.uiMinor));
	SCompilerVersion := CONCAT(SCompilerVersion, '.');
	SCompilerVersion := CONCAT(SCompilerVersion, UINT_TO_STRING(CompilerVersion.uiServicePack));
	SCompilerVersion := CONCAT(SCompilerVersion, '.');
	SCompilerVersion := CONCAT(SCompilerVersion, UINT_TO_STRING(CompilerVersion.uiPatch));	
	
	(* url *)
	IF CommonTypesAndFunctions.StrEquals(ADR(url), ADR('')) THEN
		LocalUrl := CONCAT('https://', sIpAddr);
	ELSE
		LocalUrl := url;
	END_IF
	
	SUPER^.initBaseDevice(
		Name := LEFT(THIS^.InstanceName,iSplitLocation),
		ConfigurationUrl := LocalUrl,
		Identifiers := psSerialNumber^,
		Manufacturer := WSTRING_TO_STRING(manufacturer),
		Model := WSTRING_TO_STRING(model),
		SoftwareVersion := SCompilerVersion,
		HardwareVersion := DT_TO_STRING(pstAppInfo^.dtLastChanges),
		IpAddress := sIpAddr,
		MacAddress := sMacAddr,
		availabilityTopic := availabilityTopic,			
		availabilityOnline := availabilityOnline,
		availabilityOffline := availabilityOffline,
		MqttDiscoveryPrefix := MqttDiscoveryPrefix,
		MqttDiagnosticTopic := MqttDiagnosticTopic,
		pMqttPublishQueue := pMqttPublishQueue);
		
	// Serial number diagnostic
	CreateSensorEntityWithCategory(
		Name := 'Serial number',
		Id := CONCAT(THIS^.Name,'_diag_sn'),
		Meta := '',
		StateTopic := CONCAT(MqttDiagnosticTopic, '/SN'),
		StateValue := psSerialNumber^,
		EntityCategory := 'diagnostic');
		
	// Serial number diagnostic
	CreateSensorEntityWithCategory(
		Name := 'Serial number',
		Id := CONCAT(THIS^.Name,'_diag_sn'),
		Meta := '',
		StateTopic := CONCAT(MqttDiagnosticTopic, '/SN'),
		StateValue := psSerialNumber^,
		EntityCategory := 'diagnostic');
		
	// IP address diagnostic, initial publish. done cyclic as well
	THIS^.MqttDiagnosticTopicIP := CONCAT(MqttDiagnosticTopic, '/IP');	
	MqttRefreshIP(ENQ:=TRUE, PTH:=T#0S, PTL:=T#1M);
	CreateSensorEntityWithCategory(
		Name := 'IP',
		Id := CONCAT(THIS^.Name,'_diag_ip'),
		Meta := '',
		StateTopic := THIS^.MqttDiagnosticTopicIP,
		StateValue := sIpAddr,
		EntityCategory := 'diagnostic');
		
END_IF
END_METHOD

END_FUNCTION_BLOCK

// FB_BASE_MQTT_DISCOVERY_DEVICE
{attribute 'reflection' := ''}
FUNCTION_BLOCK FB_BASE_MQTT_DISCOVERY_DEVICE
VAR
	name: STRING;
	///configuration_url
	cu: STRING;
	///connections 
	cns: ARRAY[1..2] OF ARRAY[1..2] OF STRING;
	///identifiers
	ids: STRING;
	///manufacturer
	mf: STRING;
	///model
	mdl: STRING;
	///sw_version
	sw: STRING;
	///hw_version
	hw: STRING;
	ip: STRING;
	mac: STRING;
	/// must identic to the name in the device tree
	sAppName: STRING := 'Application';
	xInit: BOOL := TRUE;
	/// object's full instance name 
	{attribute 'instance-path' := ''}
	{attribute 'noinit'}
	InstanceName: STRING;
	Startup: BOOL := TRUE;
	InitMqttDone: BOOL;
	pMqttPublishQueue: POINTER TO FB_MqttPublishQueue;
	logger: FB_MQTT_LOG;
	availabilityTopic1: STRING;
	availabilityTopic2: STRING;
	availabilityOnline: STRING;
	availabilityOffline: STRING;
	MqttDiscoveryPrefix: STRING;
	MqttDiagnosticTopic: STRING;
	MqttDiscMsgBinSens: MQTT_DISCOVERY_BINARY_SENSOR;
	MqttDiscMsgBinSensWCat: MQTT_DISCOVERY_BINARY_SENSOR_ENT_CAT;
	MqttDiscMsgCover: MQTT_DISCOVERY_COVER;
	MqttDiscMsgLightDim: MQTT_DISCOVERY_LIGHT_DIMMER;
	MqttDiscMsgLight: MQTT_DISCOVERY_LIGHT;
	MqttDiscMsgLock: MQTT_DISCOVERY_LOCK;
	MqttDiscMsgSensor: MQTT_DISCOVERY_SENSOR;
	MqttDiscMsgSensorWCat: MQTT_DISCOVERY_SENSOR_ENT_CAT;
	MqttDiscMsgSiren: MQTT_DISCOVERY_SIREN;
	MqttDiscMsgSwitch: MQTT_DISCOVERY_SWITCH;
END_VAR

{attribute 'reflection' := ''}
METHOD CreateBinarySensorEntity
VAR_INPUT
	/// default
	Name: STRING;
	Id: STRING;
	Meta: STRING;
	/// entity specific
	StateTopic: STRING;
	PayloadOn: STRING;
	PayloadOff: STRING;
	DeviceClass: STRING;
END_VAR
VAR
	EntityId: STRING(25) := 'binary_sensor';
	ComposeJSON: STRUCT_TO_JSON;
	MqttJSON: STRING(1500);
	MqttTopic: STRING(100);
END_VAR
MqttTopic := CONCAT(CONCAT(CONCAT(CONCAT(THIS^.MqttDiscoveryPrefix, EntityId),'/'), Id),'/config' );


// 	Entity related: Basis
MqttDiscMsgBinSens.name.CharString :=  name; // friendly name
MqttDiscMsgBinSens.obj_id.CharString :=  Id; 
MqttDiscMsgBinSens.uniq_id.CharString :=  Id; 

// Entity related: Specific
MqttDiscMsgBinSens.stat_t.CharString := StateTopic;
MqttDiscMsgBinSens.pl_on.CharString := PayloadOn;
MqttDiscMsgBinSens.pl_off.CharString := PayloadOff;
MqttDiscMsgBinSens.dev_cla.CharString := DeviceClass;

// Availabilty related
MqttDiscMsgBinSens.avty[1].topic.CharString := THIS^.availabilityTopic1;
MqttDiscMsgBinSens.avty[2].topic.CharString := THIS^.availabilityTopic2;
MqttDiscMsgBinSens.avty_mode.CharString := 'all';
MqttDiscMsgBinSens.pl_avail.CharString :=   THIS^.availabilityOnline;
MqttDiscMsgBinSens.pl_not_avail.CharString :=  THIS^.availabilityOffline;
MqttDiscMsgBinSens.qos.Integer := 2;

// Device related
MqttDiscMsgBinSens.dev.cu.CharString := THIS^.cu;
MqttDiscMsgBinSens.dev.name.CharString := THIS^.name;
MqttDiscMsgBinSens.dev.hw.CharString := THIS^.hw;
MqttDiscMsgBinSens.dev.ids.CharString := THIS^.ids;
MqttDiscMsgBinSens.dev.sw.CharString := THIS^.sw;
MqttDiscMsgBinSens.dev.mdl.CharString := THIS^.mdl;
MqttDiscMsgBinSens.dev.mf.CharString := THIS^.mf;
	
// Extra meta-data
IF NOT CommonTypesAndFunctions.StrEquals(str1:= ADR(meta), str2:= ADR('')) THEN
	MqttDiscMsgBinSens.meta.CharString := meta;
END_IF

ComposeJSON(
	JSONString:= ADR(MqttJSON), 
	JSONStringSize:= SIZEOF(MqttJSON),
	JSONVars:= ADR(MqttDiscMsgBinSens),
	NumberOfVars:= SIZEOF(MqttDiscMsgBinSens) / SIZEOF(JSONVAR),
	MaxLevel := 1,
);
ComposeJSON.Execute := TRUE;
ComposeJSON();

IF MqttJSON = '' THEN
	SendLogMessage(str:=CONCAT(CONCAT('ERROR ',Id), ' had empty MqttJSON'), instance := InstanceName);
ELSIF NOT (MqttJSON = '') THEN
	pMqttPublishQueue^.AddMessage(
		Payload:= MqttJSON,
		Topic := MqttTopic,
		Qos := MQTT.QoS.ExactlyOnce,
		MqttRetain := TRUE,
	);
	SendLogMessage(str:=CONCAT(CONCAT('Added ',Id), ' as MQTT dicovery'), instance := InstanceName);
END_IF
END_METHOD

{attribute 'reflection' := ''}
METHOD CreateBinarySensorEntityWithCategory
VAR_INPUT
	/// default
	Name: STRING;
	Id: STRING;
	Meta: STRING;
	/// entity specific
	StateTopic: STRING;
	PayloadOn: STRING;
	PayloadOff: STRING;
	DeviceClass: STRING;
	/// config or diagnostic
	EntityCategory: STRING;
END_VAR
VAR
	EntityId: STRING(25) := 'binary_sensor';
	ComposeJSON: STRUCT_TO_JSON;
	MqttJSON: STRING(1500);
	MqttTopic: STRING(100);
END_VAR
MqttTopic := CONCAT(CONCAT(CONCAT(CONCAT(THIS^.MqttDiscoveryPrefix, EntityId),'/'), Id),'/config' );


// 	Entity related: Basis
MqttDiscMsgBinSensWCat.name.CharString :=  name; // friendly name
MqttDiscMsgBinSensWCat.obj_id.CharString :=  Id; 
MqttDiscMsgBinSensWCat.uniq_id.CharString :=  Id; 

// Entity related: Specific
MqttDiscMsgBinSensWCat.stat_t.CharString := StateTopic;
MqttDiscMsgBinSensWCat.pl_on.CharString := PayloadOn;
MqttDiscMsgBinSensWCat.pl_off.CharString := PayloadOff;
MqttDiscMsgBinSensWCat.dev_cla.CharString := DeviceClass;
MqttDiscMsgBinSensWCat.ent_cat.CharString := EntityCategory;

// Availabilty related
MqttDiscMsgBinSensWCat.avty[1].topic.CharString := THIS^.availabilityTopic1;
MqttDiscMsgBinSensWCat.avty[2].topic.CharString := THIS^.availabilityTopic2;
MqttDiscMsgBinSensWCat.avty_mode.CharString := 'all';
MqttDiscMsgBinSensWCat.pl_avail.CharString :=   THIS^.availabilityOnline;
MqttDiscMsgBinSensWCat.pl_not_avail.CharString :=  THIS^.availabilityOffline;
MqttDiscMsgBinSensWCat.qos.Integer := 2;

// Device related
MqttDiscMsgBinSensWCat.dev.cu.CharString := THIS^.cu;
MqttDiscMsgBinSensWCat.dev.name.CharString := THIS^.name;
MqttDiscMsgBinSensWCat.dev.hw.CharString := THIS^.hw;
MqttDiscMsgBinSensWCat.dev.ids.CharString := THIS^.ids;
MqttDiscMsgBinSensWCat.dev.sw.CharString := THIS^.sw;
MqttDiscMsgBinSensWCat.dev.mdl.CharString := THIS^.mdl;
MqttDiscMsgBinSensWCat.dev.mf.CharString := THIS^.mf;
	
// Extra meta-data
IF NOT CommonTypesAndFunctions.StrEquals(str1:= ADR(meta), str2:= ADR('')) THEN
	MqttDiscMsgBinSensWCat.meta.CharString := meta;
END_IF

ComposeJSON(
	JSONString:= ADR(MqttJSON), 
	JSONStringSize:= SIZEOF(MqttJSON),
	JSONVars:= ADR(MqttDiscMsgBinSensWCat),
	NumberOfVars:= SIZEOF(MqttDiscMsgBinSensWCat) / SIZEOF(JSONVAR),
	MaxLevel := 1,
);
ComposeJSON.Execute := TRUE;
ComposeJSON();

IF MqttJSON = '' THEN
	SendLogMessage(str:=CONCAT(CONCAT('ERROR ',Id), ' had empty MqttJSON'), instance := InstanceName);
ELSIF NOT (MqttJSON = '') THEN
	pMqttPublishQueue^.AddMessage(
		Payload:= MqttJSON,
		Topic := MqttTopic,
		Qos := MQTT.QoS.ExactlyOnce,
		MqttRetain := TRUE,
	);
	SendLogMessage(str:=CONCAT(CONCAT('Added ',Id), ' as MQTT dicovery'), instance := InstanceName);
END_IF
END_METHOD

METHOD CreateCoverEntity
VAR_INPUT
	/// default
	Name: STRING;
	Id: STRING;
	Meta: STRING;
	/// entity specific
	CommandTopic: STRING;
	PayloadOpen: STRING;
	PayloadClose: STRING;
	PayloadStop: STRING;
	StateTopic: STRING;
	StateOpen: STRING;
	StateClosed: STRING;
	Deviceclass: STRING;
END_VAR
VAR
	EntityId: STRING(25) := 'cover';
	ComposeJSON: STRUCT_TO_JSON;
	MqttJSON: STRING(1500);
	MqttTopic: STRING(100);
END_VAR
MqttTopic := CONCAT(CONCAT(CONCAT(CONCAT(THIS^.MqttDiscoveryPrefix, EntityId),'/'), Id),'/config' );

// 	Entity related: Basis
MqttDiscMsgCover.name.CharString :=  name; // friendly name
MqttDiscMsgCover.obj_id.CharString :=  Id; 
MqttDiscMsgCover.uniq_id.CharString :=  Id; 

// Entity related: Specific
MqttDiscMsgCover.cmd_t.CharString := CommandTopic;
MqttDiscMsgCover.pl_open.CharString := PayloadOpen;
MqttDiscMsgCover.pl_cls.CharString := PayloadClose;
MqttDiscMsgCover.pl_stop.CharString := PayloadStop;
MqttDiscMsgCover.stat_t.CharString := StateTopic;
MqttDiscMsgCover.stat_open.CharString := StateOpen;
MqttDiscMsgCover.stat_clsd.CharString := StateClosed;
MqttDiscMsgCover.opt.Boolean := FALSE;
MqttDiscMsgCover.dev_cla.CharString := Deviceclass;

// Availabilty related
MqttDiscMsgCover.avty[1].topic.CharString := THIS^.availabilityTopic1;
MqttDiscMsgCover.avty[2].topic.CharString := THIS^.availabilityTopic2;
MqttDiscMsgCover.avty_mode.CharString := 'all';
MqttDiscMsgCover.pl_avail.CharString :=   THIS^.availabilityOnline;
MqttDiscMsgCover.pl_not_avail.CharString :=  THIS^.availabilityOffline;
MqttDiscMsgCover.qos.Integer := 2;

// Device related
MqttDiscMsgCover.dev.cu.CharString := THIS^.cu;
MqttDiscMsgCover.dev.name.CharString := THIS^.name;
MqttDiscMsgCover.dev.hw.CharString := THIS^.hw;
MqttDiscMsgCover.dev.ids.CharString := THIS^.ids;
MqttDiscMsgCover.dev.sw.CharString := THIS^.sw;
MqttDiscMsgCover.dev.mdl.CharString := THIS^.mdl;
MqttDiscMsgCover.dev.mf.CharString := THIS^.mf;
	
// Extra meta-data
IF NOT CommonTypesAndFunctions.StrEquals(str1:= ADR(meta), str2:= ADR('')) THEN
	MqttDiscMsgCover.meta.CharString := meta;
END_IF

ComposeJSON(
	JSONString:= ADR(MqttJSON), 
	JSONStringSize:= SIZEOF(MqttJSON),
	JSONVars:= ADR(MqttDiscMsgCover),
	NumberOfVars:= SIZEOF(MqttDiscMsgCover) / SIZEOF(JSONVAR),
	MaxLevel := 1,
);
ComposeJSON.Execute := TRUE;
ComposeJSON();

IF MqttJSON = '' THEN
	SendLogMessage(str:=CONCAT(CONCAT('ERROR ',Id), ' had empty MqttJSON'), instance := InstanceName);
ELSIF NOT (MqttJSON = '') THEN
	pMqttPublishQueue^.AddMessage(
		Payload:= MqttJSON,
		Topic := MqttTopic,
		Qos := MQTT.QoS.ExactlyOnce,
		MqttRetain := TRUE,
	);
	SendLogMessage(str:=CONCAT(CONCAT('Added ',Id), ' as MQTT dicovery'), instance := InstanceName);
END_IF
END_METHOD

METHOD CreateLightDimmerEntity
VAR_INPUT
	/// default
	Name: STRING;
	Id: STRING;
	Meta: STRING;
	/// entity specific
	CommandTopic: STRING;
	PayloadOn: STRING;
	PayloadOff: STRING;
	StateTopic: STRING;
	BrightnessCommandTopic: STRING;
	BrightnessStateTopic: STRING;
	BrightnessScale: INT;
	/// dmx specific
	DmxChannel: INT := 0;
	DmxWidth: INT := 0;
	DmxUniverse: INT := 0;
END_VAR
VAR
	EntityId: STRING(25) := 'light';
	ComposeJSON: STRUCT_TO_JSON;
	MqttJSON: STRING(1500);
	MqttTopic: STRING(100);
END_VAR
MqttTopic := CONCAT(CONCAT(CONCAT(CONCAT(THIS^.MqttDiscoveryPrefix, EntityId),'/'), Id),'/config' );

// 	Entity related: Basis
MqttDiscMsgLightDim.name.CharString :=  name; // friendly name
MqttDiscMsgLightDim.obj_id.CharString :=  Id; 
MqttDiscMsgLightDim.uniq_id.CharString :=  Id; 

// Entity related: Specific
MqttDiscMsgLightDim.cmd_t.CharString := CommandTopic;
MqttDiscMsgLightDim.pl_on.CharString := PayloadOn;
MqttDiscMsgLightDim.pl_off.CharString := PayloadOff;
MqttDiscMsgLightDim.stat_t.CharString := StateTopic;
MqttDiscMsgLightDim.opt.Boolean := FALSE;

MqttDiscMsgLightDim.bri_cmd_t.CharString := BrightnessCommandTopic;
MqttDiscMsgLightDim.bri_stat_t.CharString := BrightnessStateTopic;
MqttDiscMsgLightDim.bri_scl.Integer := BrightnessScale;
MqttDiscMsgLightDim.on_cmd_type.CharString := 'last';

MqttDiscMsgLightDim.dmxChannel.Integer := DmxChannel;
MqttDiscMsgLightDim.dmxWidth.Integer := DmxWidth;
MqttDiscMsgLightDim.dmxUniverse.Integer := DmxUniverse;

// Availabilty related
MqttDiscMsgLightDim.avty[1].topic.CharString := THIS^.availabilityTopic1;
MqttDiscMsgLightDim.avty[2].topic.CharString := THIS^.availabilityTopic2;
MqttDiscMsgLightDim.avty_mode.CharString := 'all';
MqttDiscMsgLightDim.pl_avail.CharString :=   THIS^.availabilityOnline;
MqttDiscMsgLightDim.pl_not_avail.CharString :=  THIS^.availabilityOffline;
MqttDiscMsgLightDim.qos.Integer := 2;

// Device related
MqttDiscMsgLightDim.dev.cu.CharString := THIS^.cu;
MqttDiscMsgLightDim.dev.name.CharString := THIS^.name;
MqttDiscMsgLightDim.dev.hw.CharString := THIS^.hw;
MqttDiscMsgLightDim.dev.ids.CharString := THIS^.ids;
MqttDiscMsgLightDim.dev.sw.CharString := THIS^.sw;
MqttDiscMsgLightDim.dev.mdl.CharString := THIS^.mdl;
MqttDiscMsgLightDim.dev.mf.CharString := THIS^.mf;
	
// Extra meta-data
IF NOT CommonTypesAndFunctions.StrEquals(str1:= ADR(meta), str2:= ADR('')) THEN
	MqttDiscMsgLightDim.meta.CharString := meta;
END_IF

ComposeJSON(
	JSONString:= ADR(MqttJSON), 
	JSONStringSize:= SIZEOF(MqttJSON),
	JSONVars:= ADR(MqttDiscMsgLightDim),
	NumberOfVars:= SIZEOF(MqttDiscMsgLightDim) / SIZEOF(JSONVAR),
	MaxLevel := 1,
);
ComposeJSON.Execute := TRUE;
ComposeJSON();

IF MqttJSON = '' THEN
	SendLogMessage(str:=CONCAT(CONCAT('ERROR ',Id), ' had empty MqttJSON'), instance := InstanceName);
ELSIF NOT (MqttJSON = '') THEN
	pMqttPublishQueue^.AddMessage(
		Payload:= MqttJSON,
		Topic := MqttTopic,
		Qos := MQTT.QoS.ExactlyOnce,
		MqttRetain := TRUE,
	);
	SendLogMessage(str:=CONCAT(CONCAT('Added ',Id), ' as MQTT dicovery'), instance := InstanceName);
END_IF
END_METHOD

METHOD CreateLightEntity
VAR_INPUT
	/// default
	Name: STRING;
	Id: STRING;
	Meta: STRING;
	/// entity specific
	CommandTopic: STRING;
	PayloadOn: STRING;
	PayloadOff: STRING;
	StateTopic: STRING;
END_VAR
VAR
	EntityId: STRING(25) := 'light';
	ComposeJSON: STRUCT_TO_JSON;
	MqttJSON: STRING(1500);
	MqttTopic: STRING(100);
END_VAR
MqttTopic := CONCAT(CONCAT(CONCAT(CONCAT(THIS^.MqttDiscoveryPrefix, EntityId),'/'), Id),'/config' );

// 	Entity related: Basis
MqttDiscMsgLight.name.CharString :=  name; // friendly name
MqttDiscMsgLight.obj_id.CharString :=  Id; 
MqttDiscMsgLight.uniq_id.CharString :=  Id; 

// Entity related: Specific
MqttDiscMsgLight.cmd_t.CharString := CommandTopic;
MqttDiscMsgLight.pl_on.CharString := PayloadOn;
MqttDiscMsgLight.pl_off.CharString := PayloadOff;
MqttDiscMsgLight.stat_t.CharString := StateTopic;
MqttDiscMsgLight.opt.Boolean := FALSE;

// Availabilty related
MqttDiscMsgLight.avty[1].topic.CharString := THIS^.availabilityTopic1;
MqttDiscMsgLight.avty[2].topic.CharString := THIS^.availabilityTopic2;
MqttDiscMsgLight.avty_mode.CharString := 'all';
MqttDiscMsgLight.pl_avail.CharString :=   THIS^.availabilityOnline;
MqttDiscMsgLight.pl_not_avail.CharString :=  THIS^.availabilityOffline;
MqttDiscMsgLight.qos.Integer := 2;

// Device related
MqttDiscMsgLight.dev.cu.CharString := THIS^.cu;
MqttDiscMsgLight.dev.name.CharString := THIS^.name;
MqttDiscMsgLight.dev.hw.CharString := THIS^.hw;
MqttDiscMsgLight.dev.ids.CharString := THIS^.ids;
MqttDiscMsgLight.dev.sw.CharString := THIS^.sw;
MqttDiscMsgLight.dev.mdl.CharString := THIS^.mdl;
MqttDiscMsgLight.dev.mf.CharString := THIS^.mf;
	
// Extra meta-data
IF NOT CommonTypesAndFunctions.StrEquals(str1:= ADR(meta), str2:= ADR('')) THEN
	MqttDiscMsgLight.meta.CharString := meta;
END_IF

ComposeJSON(
	JSONString:= ADR(MqttJSON), 
	JSONStringSize:= SIZEOF(MqttJSON),
	JSONVars:= ADR(MqttDiscMsgLight),
	NumberOfVars:= SIZEOF(MqttDiscMsgLight) / SIZEOF(JSONVAR),
	MaxLevel := 1,
);
ComposeJSON.Execute := TRUE;
ComposeJSON();

IF MqttJSON = '' THEN
	SendLogMessage(str:=CONCAT(CONCAT('ERROR ',Id), ' had empty MqttJSON'), instance := InstanceName);
ELSIF NOT (MqttJSON = '') THEN
	pMqttPublishQueue^.AddMessage(
		Payload:= MqttJSON,
		Topic := MqttTopic,
		Qos := MQTT.QoS.ExactlyOnce,
		MqttRetain := TRUE,
	);
	SendLogMessage(str:=CONCAT(CONCAT('Added ',Id), ' as MQTT dicovery'), instance := InstanceName);
END_IF
END_METHOD

METHOD CreateLockEntity
VAR_INPUT
	/// default
	Name: STRING;
	Id: STRING;
	Meta: STRING;
	/// entity specific
	CommandTopic: STRING;
	PayloadLock: STRING;
	PayloadUnlock: STRING;
	StateTopic: STRING;
	StateLocked: STRING;
	StateUnlocked: STRING;
END_VAR
VAR
	EntityId: STRING(25) := 'lock';
	ComposeJSON: STRUCT_TO_JSON;
	MqttJSON: STRING(1500);
	MqttTopic: STRING(100);
END_VAR
MqttTopic := CONCAT(CONCAT(CONCAT(CONCAT(THIS^.MqttDiscoveryPrefix, EntityId),'/'), Id),'/config' );

// 	Entity related: Basis
MqttDiscMsgLock.name.CharString :=  name; // friendly name
MqttDiscMsgLock.obj_id.CharString :=  Id; 
MqttDiscMsgLock.uniq_id.CharString :=  Id; 

// Entity related: Specific
MqttDiscMsgLock.cmd_t.CharString := CommandTopic;
MqttDiscMsgLock.pl_lock.CharString := PayloadLock;
MqttDiscMsgLock.pl_unlk.CharString := PayloadUnlock;
MqttDiscMsgLock.stat_t.CharString := StateTopic;
MqttDiscMsgLock.stat_locked.CharString := StateLocked;
MqttDiscMsgLock.stat_unlocked.CharString := StateUnlocked;
MqttDiscMsgLock.opt.Boolean := FALSE;

// Availabilty related
MqttDiscMsgLock.avty[1].topic.CharString := THIS^.availabilityTopic1;
MqttDiscMsgLock.avty[2].topic.CharString := THIS^.availabilityTopic2;
MqttDiscMsgLock.avty_mode.CharString := 'all';
MqttDiscMsgLock.pl_avail.CharString :=   THIS^.availabilityOnline;
MqttDiscMsgLock.pl_not_avail.CharString :=  THIS^.availabilityOffline;
MqttDiscMsgLock.qos.Integer := 2;

// Device related
MqttDiscMsgLock.dev.cu.CharString := THIS^.cu;
MqttDiscMsgLock.dev.name.CharString := THIS^.name;
MqttDiscMsgLock.dev.hw.CharString := THIS^.hw;
MqttDiscMsgLock.dev.ids.CharString := THIS^.ids;
MqttDiscMsgLock.dev.sw.CharString := THIS^.sw;
MqttDiscMsgLock.dev.mdl.CharString := THIS^.mdl;
MqttDiscMsgLock.dev.mf.CharString := THIS^.mf;
	
// Extra meta-data
IF NOT CommonTypesAndFunctions.StrEquals(str1:= ADR(meta), str2:= ADR('')) THEN
	MqttDiscMsgLock.meta.CharString := meta;
END_IF

ComposeJSON(
	JSONString:= ADR(MqttJSON), 
	JSONStringSize:= SIZEOF(MqttJSON),
	JSONVars:= ADR(MqttDiscMsgLock),
	NumberOfVars:= SIZEOF(MqttDiscMsgLock) / SIZEOF(JSONVAR),
	MaxLevel := 1,
);
ComposeJSON.Execute := TRUE;
ComposeJSON();

IF MqttJSON = '' THEN
	SendLogMessage(str:=CONCAT(CONCAT('ERROR ',Id), ' had empty MqttJSON'), instance := InstanceName);
ELSIF NOT (MqttJSON = '') THEN
	pMqttPublishQueue^.AddMessage(
		Payload:= MqttJSON,
		Topic := MqttTopic,
		Qos := MQTT.QoS.ExactlyOnce,
		MqttRetain := TRUE,
	);
	SendLogMessage(str:=CONCAT(CONCAT('Added ',Id), ' as MQTT dicovery'), instance := InstanceName);
END_IF
END_METHOD

METHOD CreateSensorEntity
VAR_INPUT
	/// default
	Name: STRING;
	Id: STRING;
	Meta: STRING;
	/// entity specific
	StateTopic: STRING;
	ExpiryAfter: INT := 0;
END_VAR
VAR
	EntityId: STRING(25) := 'sensor';
	ComposeJSON: STRUCT_TO_JSON;
	MqttJSON: STRING(1500);
	MqttTopic: STRING(100);
END_VAR
MqttTopic := CONCAT(CONCAT(CONCAT(CONCAT(THIS^.MqttDiscoveryPrefix, EntityId),'/'), Id),'/config' );

// 	Entity related: Basis
MqttDiscMsgSensor.name.CharString :=  name; // friendly name
MqttDiscMsgSensor.obj_id.CharString :=  Id; 
MqttDiscMsgSensor.uniq_id.CharString :=  Id; 

// Entity related: Specific
//MqttDiscoverySensorMessage.ic.CharString := Icon;
MqttDiscMsgSensor.stat_t.CharString := StateTopic;
MqttDiscMsgSensor.exp_aft.Integer := ExpiryAfter;

// Availabilty related
MqttDiscMsgSensor.avty[1].topic.CharString := THIS^.availabilityTopic1;
MqttDiscMsgSensor.avty[2].topic.CharString := THIS^.availabilityTopic2;
MqttDiscMsgSensor.avty_mode.CharString := 'all';
MqttDiscMsgSensor.pl_avail.CharString :=   THIS^.availabilityOnline;
MqttDiscMsgSensor.pl_not_avail.CharString :=  THIS^.availabilityOffline;
MqttDiscMsgSensor.qos.Integer := 2;

// Device related
MqttDiscMsgSensor.dev.cu.CharString := THIS^.cu;
MqttDiscMsgSensor.dev.name.CharString := THIS^.name;
MqttDiscMsgSensor.dev.hw.CharString := THIS^.hw;
MqttDiscMsgSensor.dev.ids.CharString := THIS^.ids;
MqttDiscMsgSensor.dev.sw.CharString := THIS^.sw;
MqttDiscMsgSensor.dev.mdl.CharString := THIS^.mdl;
MqttDiscMsgSensor.dev.mf.CharString := THIS^.mf;
	
// Extra meta-data
IF NOT CommonTypesAndFunctions.StrEquals(str1:= ADR(meta), str2:= ADR('')) THEN
	MqttDiscMsgSensor.meta.CharString := meta;
END_IF

ComposeJSON(
	JSONString:= ADR(MqttJSON), 
	JSONStringSize:= SIZEOF(MqttJSON),
	JSONVars:= ADR(MqttDiscMsgSensor),
	NumberOfVars:= SIZEOF(MqttDiscMsgSensor) / SIZEOF(JSONVAR),
	MaxLevel := 1,
);
ComposeJSON.Execute := TRUE;
ComposeJSON();

IF MqttJSON = '' THEN
	SendLogMessage(str:=CONCAT(CONCAT('ERROR ',Id), ' had empty MqttJSON'), instance := InstanceName);
ELSIF NOT (MqttJSON = '') THEN
	pMqttPublishQueue^.AddMessage(
		Payload:= MqttJSON,
		Topic := MqttTopic,
		Qos := MQTT.QoS.ExactlyOnce,
		MqttRetain := TRUE,
	);
	SendLogMessage(str:=CONCAT(CONCAT('Added ',Id), ' as MQTT dicovery'), instance := InstanceName);
END_IF
END_METHOD

METHOD CreateSensorEntityWithCategory
VAR_INPUT
	/// default
	Name: STRING;
	Id: STRING;
	Meta: STRING;
	/// entity specific
	StateTopic: STRING;
	StateValue: STRING := '';
	/// config or diagnostic
	EntityCategory: STRING;
	ExpiryAfter: INT := 0;
END_VAR
VAR
	EntityId: STRING(25) := 'sensor';
	ComposeJSON: STRUCT_TO_JSON;
	MqttJSON: STRING(1500);
	MqttTopic: STRING(100);
END_VAR
MqttTopic := CONCAT(CONCAT(CONCAT(CONCAT(THIS^.MqttDiscoveryPrefix, EntityId),'/'), Id),'/config' );

// 	Entity related: Basis
MqttDiscMsgSensorWCat.name.CharString :=  name; // friendly name
MqttDiscMsgSensorWCat.obj_id.CharString :=  Id; 
MqttDiscMsgSensorWCat.uniq_id.CharString :=  Id; 

// Entity related: Specific
//MqttDiscoverySensorMessage.ic.CharString := Icon;
MqttDiscMsgSensorWCat.stat_t.CharString := StateTopic;
MqttDiscMsgSensorWCat.exp_aft.Integer := ExpiryAfter;
MqttDiscMsgSensorWCat.ent_cat.CharString := EntityCategory;

// Availabilty related
MqttDiscMsgSensorWCat.avty[1].topic.CharString := THIS^.availabilityTopic1;
MqttDiscMsgSensorWCat.avty[2].topic.CharString := THIS^.availabilityTopic2;
MqttDiscMsgSensorWCat.avty_mode.CharString := 'all';
MqttDiscMsgSensorWCat.pl_avail.CharString :=   THIS^.availabilityOnline;
MqttDiscMsgSensorWCat.pl_not_avail.CharString :=  THIS^.availabilityOffline;
MqttDiscMsgSensorWCat.qos.Integer := 2;

// Device related
MqttDiscMsgSensorWCat.dev.cu.CharString := THIS^.cu;
MqttDiscMsgSensorWCat.dev.name.CharString := THIS^.name;
MqttDiscMsgSensorWCat.dev.hw.CharString := THIS^.hw;
MqttDiscMsgSensorWCat.dev.ids.CharString := THIS^.ids;
MqttDiscMsgSensorWCat.dev.sw.CharString := THIS^.sw;
MqttDiscMsgSensorWCat.dev.mdl.CharString := THIS^.mdl;
MqttDiscMsgSensorWCat.dev.mf.CharString := THIS^.mf;
	
// Extra meta-data
IF NOT CommonTypesAndFunctions.StrEquals(str1:= ADR(meta), str2:= ADR('')) THEN
	MqttDiscMsgSensorWCat.meta.CharString := meta;
END_IF

ComposeJSON(
	JSONString:= ADR(MqttJSON), 
	JSONStringSize:= SIZEOF(MqttJSON),
	JSONVars:= ADR(MqttDiscMsgSensorWCat),
	NumberOfVars:= SIZEOF(MqttDiscMsgSensorWCat) / SIZEOF(JSONVAR),
	MaxLevel := 1,
);
ComposeJSON.Execute := TRUE;
ComposeJSON();

IF MqttJSON = '' THEN
	SendLogMessage(str:=CONCAT(CONCAT('ERROR ',Id), ' had empty MqttJSON'), instance := InstanceName);
ELSIF NOT (MqttJSON = '') THEN
	pMqttPublishQueue^.AddMessage(
		Payload:= MqttJSON,
		Topic := MqttTopic,
		Qos := MQTT.QoS.ExactlyOnce,
		MqttRetain := TRUE,
	);
	IF NOT (StateValue = '') THEN		
		pMqttPublishQueue^.AddMessage(
			Payload:= StateValue,
			Topic := StateTopic,
			Qos := MQTT.QoS.ExactlyOnce,
			MqttRetain := TRUE,
		);
	END_IF
	
	SendLogMessage(str:=CONCAT(CONCAT('Added ',Id), ' as MQTT dicovery'), instance := InstanceName);
END_IF
END_METHOD

METHOD CreateSirenEntity
VAR_INPUT
	/// default
	Name: STRING;
	Id: STRING;
	Meta: STRING;
	/// entity specific
	CommandTopic: STRING;
	PayloadOn: STRING;
	PayloadOff: STRING;
	StateTopic: STRING;
	StateOnPayload: STRING;
	StateOffPayload: STRING;
END_VAR
VAR
	EntityId: STRING(25) := 'siren';
	ComposeJSON: STRUCT_TO_JSON;
	MqttJSON: STRING(1500);
	MqttTopic: STRING(100);
END_VAR
MqttTopic := CONCAT(CONCAT(CONCAT(CONCAT(THIS^.MqttDiscoveryPrefix, EntityId),'/'), Id),'/config' );

// 	Entity related: Basis
MqttDiscMsgSiren.name.CharString :=  name; // friendly name
MqttDiscMsgSiren.obj_id.CharString :=  Id; 
MqttDiscMsgSiren.uniq_id.CharString :=  Id; 

// Entity related: Specific
MqttDiscMsgSiren.cmd_t.CharString := CommandTopic;
MqttDiscMsgSiren.pl_on.CharString := PayloadOn;
MqttDiscMsgSiren.pl_off.CharString := PayloadOff;
MqttDiscMsgSiren.stat_t.CharString := StateTopic;
MqttDiscMsgSiren.stat_on.CharString := StateOnPayload;
MqttDiscMsgSiren.stat_off.CharString := StateOffPayload;
MqttDiscMsgSiren.opt.Boolean := FALSE;

// Availabilty related
MqttDiscMsgSiren.avty[1].topic.CharString := THIS^.availabilityTopic1;
MqttDiscMsgSiren.avty[2].topic.CharString := THIS^.availabilityTopic2;
MqttDiscMsgSiren.avty_mode.CharString := 'all';
MqttDiscMsgSiren.pl_avail.CharString :=   THIS^.availabilityOnline;
MqttDiscMsgSiren.pl_not_avail.CharString :=  THIS^.availabilityOffline;
MqttDiscMsgSiren.qos.Integer := 2;


// Device related
MqttDiscMsgSiren.dev.cu.CharString := THIS^.cu;
MqttDiscMsgSiren.dev.name.CharString := THIS^.name;
MqttDiscMsgSiren.dev.hw.CharString := THIS^.hw;
MqttDiscMsgSiren.dev.ids.CharString := THIS^.ids;
MqttDiscMsgSiren.dev.sw.CharString := THIS^.sw;
MqttDiscMsgSiren.dev.mdl.CharString := THIS^.mdl;
MqttDiscMsgSiren.dev.mf.CharString := THIS^.mf;
	
// Extra meta-data
IF NOT CommonTypesAndFunctions.StrEquals(str1:= ADR(meta), str2:= ADR('')) THEN
	MqttDiscMsgSiren.meta.CharString := meta;
END_IF

ComposeJSON(
	JSONString:= ADR(MqttJSON), 
	JSONStringSize:= SIZEOF(MqttJSON),
	JSONVars:= ADR(MqttDiscMsgSiren),
	NumberOfVars:= SIZEOF(MqttDiscMsgSiren) / SIZEOF(JSONVAR),
	MaxLevel := 1,
);
ComposeJSON.Execute := TRUE;
ComposeJSON();

IF MqttJSON = '' THEN
	SendLogMessage(str:=CONCAT(CONCAT('ERROR ',Id), ' had empty MqttJSON'), instance := InstanceName);
ELSIF NOT (MqttJSON = '') THEN
	pMqttPublishQueue^.AddMessage(
		Payload:= MqttJSON,
		Topic := MqttTopic,
		Qos := MQTT.QoS.ExactlyOnce,
		MqttRetain := TRUE,
	);
	SendLogMessage(str:=CONCAT(CONCAT('Added ',Id), ' as MQTT dicovery'), instance := InstanceName);
END_IF
END_METHOD

METHOD CreateSwitchEntity
VAR_INPUT
	/// default
	Name: STRING;
	Id: STRING;
	Meta: STRING;
	/// entity specific
	CommandTopic: STRING;
	PayloadOn: STRING;
	PayloadOff: STRING;
	StateTopic: STRING;
	StateOnPayload: STRING;
	StateOffPayload: STRING;
	DeviceClass: STRING;
END_VAR
VAR
	EntityId: STRING(25) := 'switch';
	ComposeJSON: STRUCT_TO_JSON;
	MqttJSON: STRING(1500);
	MqttTopic: STRING(100);
END_VAR
MqttTopic := CONCAT(CONCAT(CONCAT(CONCAT(THIS^.MqttDiscoveryPrefix, EntityId),'/'), Id),'/config' );

// 	Entity related: Basis
MqttDiscMsgSwitch.name.CharString :=  name; // friendly name
MqttDiscMsgSwitch.obj_id.CharString :=  Id; 
MqttDiscMsgSwitch.uniq_id.CharString :=  Id; 

// Entity related: Specific
MqttDiscMsgSwitch.cmd_t.CharString := CommandTopic;
MqttDiscMsgSwitch.pl_on.CharString := PayloadOn;
MqttDiscMsgSwitch.pl_off.CharString := PayloadOff;
MqttDiscMsgSwitch.stat_t.CharString := StateTopic;
MqttDiscMsgSwitch.stat_on.CharString := StateOnPayload;
MqttDiscMsgSwitch.stat_off.CharString := StateOffPayload;
MqttDiscMsgSwitch.opt.Boolean := FALSE;
MqttDiscMsgSwitch.dev_cla.CharString := DeviceClass;

// Availabilty related
MqttDiscMsgSwitch.avty[1].topic.CharString := THIS^.availabilityTopic1;
MqttDiscMsgSwitch.avty[2].topic.CharString := THIS^.availabilityTopic2;
MqttDiscMsgSwitch.avty_mode.CharString := 'all';
MqttDiscMsgSwitch.pl_avail.CharString :=   THIS^.availabilityOnline;
MqttDiscMsgSwitch.pl_not_avail.CharString :=  THIS^.availabilityOffline;
MqttDiscMsgSwitch.qos.Integer := 2;

// Device related
MqttDiscMsgSwitch.dev.cu.CharString := THIS^.cu;
MqttDiscMsgSwitch.dev.name.CharString := THIS^.name;
MqttDiscMsgSwitch.dev.hw.CharString := THIS^.hw;
MqttDiscMsgSwitch.dev.ids.CharString := THIS^.ids;
MqttDiscMsgSwitch.dev.sw.CharString := THIS^.sw;
MqttDiscMsgSwitch.dev.mdl.CharString := THIS^.mdl;
MqttDiscMsgSwitch.dev.mf.CharString := THIS^.mf;
	
// Extra meta-data
IF NOT CommonTypesAndFunctions.StrEquals(str1:= ADR(meta), str2:= ADR('')) THEN
	MqttDiscMsgSwitch.meta.CharString := meta;
END_IF

ComposeJSON(
	JSONString:= ADR(MqttJSON), 
	JSONStringSize:= SIZEOF(MqttJSON),
	JSONVars:= ADR(MqttDiscMsgSwitch),
	NumberOfVars:= SIZEOF(MqttDiscMsgSwitch) / SIZEOF(JSONVAR),
	MaxLevel := 1,
);
ComposeJSON.Execute := TRUE;
ComposeJSON();

IF MqttJSON = '' THEN
	SendLogMessage(str:=CONCAT(CONCAT('ERROR ',Id), ' had empty MqttJSON'), instance := InstanceName);
ELSIF NOT (MqttJSON = '') THEN
	pMqttPublishQueue^.AddMessage(
		Payload:= MqttJSON,
		Topic := MqttTopic,
		Qos := MQTT.QoS.ExactlyOnce,
		MqttRetain := TRUE,
	);
	SendLogMessage(str:=CONCAT(CONCAT('Added ',Id), ' as MQTT dicovery'), instance := InstanceName);
END_IF
END_METHOD

METHOD initBaseDevice
VAR_INPUT
	Name: STRING;
	ConfigurationUrl: STRING;
	Identifiers: STRING;
	Manufacturer: STRING;
	Model: STRING;
	SoftwareVersion: STRING;
	HardwareVersion: STRING;
	IpAddress: STRING := '';
	MacAddress: STRING := '';
	availabilityTopic: STRING;
	availabilityTopic2: STRING := '';
	availabilityOnline: STRING;
	availabilityOffline: STRING;
	MqttDiscoveryPrefix: STRING;
	MqttDiagnosticTopic: STRING;
	pMqttPublishQueue: POINTER TO FB_MqttPublishQueue;
END_VAR
THIS^.availabilityTopic1 := availabilityTopic;

IF CommonTypesAndFunctions.StrEquals(str1:= ADR(availabilityTopic2), str2:= ADR('')) THEN
	THIS^.availabilityTopic2 := availabilityTopic;
ELSE
	THIS^.availabilityTopic2 := availabilityTopic2;
END_IF

THIS^.availabilityOnline := availabilityOnline;
THIS^.availabilityOffline := availabilityOffline;
THIS^.pMqttPublishQueue := pMqttPublishQueue;
THIS^.MqttDiscoveryPrefix := MqttDiscoveryPrefix;
THIS^.MqttDiagnosticTopic := MqttDiagnosticTopic;

THIS^.name := Name;
THIS^.cu:= ConfigurationUrl;
THIS^.ids:= Identifiers;
THIS^.mf:= Manufacturer;
THIS^.mdl:= Model;
THIS^.hw:= HardwareVersion;
THIS^.sw:= SoftwareVersion;
THIS^.ip := IpAddress;
THIS^.mac := MacAddress;

//Create a diagnostics availability binary sensor
CreateBinarySensorEntityWithCategory(
	Name := 'Availability',
	Id := CONCAT(THIS^.Name,'_diag_availability'),
	Meta := '',
	StateTopic := availabilityTopic,
	PayloadOn := availabilityOnline,
	PayloadOff := availabilityOffline,
	DeviceClass := 'CONNECTIVITY',
	EntityCategory := 'diagnostic');
	
//Logger
CreateSensorEntityWithCategory(
		Name := 'Log',
		Id := CONCAT(THIS^.Name,'_diag_log'),
		Meta := '',
		StateTopic := CONCAT(MqttDiagnosticTopic, '/Log'),
		EntityCategory := 'diagnostic');
	
// MAC address
IF NOT(MacAddress = '') THEN
	CreateSensorEntityWithCategory(
		Name := 'MAC',
		Id := CONCAT(THIS^.Name,'_diag_mac'),
		Meta := '',
		StateTopic := CONCAT(MqttDiagnosticTopic, '/MAC'),
		StateValue := MacAddress,
		EntityCategory := 'diagnostic');	
END_IF
END_METHOD

METHOD SendLogMessage : BOOL
VAR_INPUT
	str: STRING(128);
	instance: STRING := '';
END_VAR
pMqttPublishQueue^.AddMessage(
	Payload:= CONCAT(CONCAT(instance,' | '),str),
	Topic := CONCAT(MqttDiagnosticTopic, '/Log'),
	Qos := 1,
	MqttRetain := TRUE
);
END_METHOD

END_FUNCTION_BLOCK

// FB_MQTT_LOG
FUNCTION_BLOCK FB_MQTT_LOG EXTENDS FB_MQTT_BASE
VAR
	/// should have a dot in the name
	InstancePath: STRING := '.plc_log';
	MqttDiscoveryMessage: MQTT_DISCOVERY_SENSOR;
END_VAR

METHOD InitMqtt
VAR_INPUT
	MQTTPublishPrefix: POINTER TO STRING;
	pMqttPublishQueue: POINTER TO FB_MqttPublishQueue;
	MqttQos: MQTT.QoS := MQTT.QoS.ExactlyOnce;
	MqttRetain: BOOL := FALSE;
END_VAR
SUPER^._InstancePath := THIS^.InstancePath; // Due to reflection its location is important

(*pass trough*)
THIS^.pMqttPublishQueue := pMqttPublishQueue;
THIS^.MqttPublishTopicPrefix:=MQTTPublishPrefix;
THIS^.pMqttPublishQueue:=pMqttPublishQueue;

THIS^.MqttQos := MqttQos;
THIS^.MqttRetain := MqttRetain;

SUPER^.InitBaseMqtt();
END_METHOD

METHOD InitMqttDiscovery
VAR_INPUT
	Device: POINTER TO FB_PLC_MQTT_DISCOVERY_DEVICE;
	Name: STRING(255) := 'plc_log';
	overruleId: STRING(255) := '';
	meta: STRING(255) := '';
END_VAR
VAR
	id: STRING(255);
END_VAR
IF InitMqttDone AND NOT initMqttDiscoveryDone THEN
	
	IF CommonTypesAndFunctions.StrEquals(str1:= ADR(overruleId), str2:= ADR('')) THEN
		id := CONCAT(CONCAT(THIS^.DeviceName,'_'), THIS^.InstanceNamePt^); // 'FB_DI_PB_003'
	ELSE
		id := overruleId; // 'MY_PH_GND_HALL_01'
	END_IF	
	
	Device^.CreateSensorEntity(
		Name := name,
		Id := id,
		Meta := meta,
		StateTopic := THIS^.MQTTPublishTopic);

	initMqttDiscoveryDone := TRUE;
END_IF
END_METHOD

METHOD send
VAR_INPUT
	str: STRING(128);
	instance: STRING := '';
END_VAR
IF InitMqttDone THEN
	pMqttPublishQueue^.AddMessage(
		Payload:= CONCAT(CONCAT(instance,' | '),str),
		Topic := THIS^.MQTTPublishTopic,
		Qos := 1,
		MqttRetain := TRUE
	);
END_IF
END_METHOD

END_FUNCTION_BLOCK

// FB_INPUT_PUSHBUTTON_DIMMER_MQTT
{attribute 'reflection' := ''}
FUNCTION_BLOCK FB_INPUT_PUSHBUTTON_DIMMER_MQTT
VAR_INPUT
	PB: BOOL;
	SET: BOOL;
	VAL: BYTE;
	RST: BOOL;
END_VAR
VAR_OUTPUT
	DIM: BYTE;
	DBL: BOOL;
	Q: BOOL;
	SINGLE: BOOL;
	DOUBLE: BOOL;
	LONG: BOOL;
	P_LONG: BOOL;
END_VAR
VAR
	/// object's full instance name 
	{attribute 'noinit'}
	{attribute 'instance-path' := ''}
	InstanceName: STRING;
	InitMqttDone: BOOL;
	MqttPublishTopicPrefix: POINTER TO STRING;
	MqttPublishTopicSuffix: STRING(50);
	pMqttPublishQueue: POINTER TO FB_MqttPublishQueue;
	FB_DIMMER: OSCAT_BUILDING.DIMM_I;
	OutputDimmer: BOOL;
	Qos_Dimm: MQTT.QoS;
	Delta_Dimm: INT;
	FB_DETECTPUSH: OSCAT_BUILDING.CLICK_MODE;
	P_LONG_R_TRIG: Standard.R_TRIG;
	P_LONG_F_TRIG: Standard.F_TRIG;
	/// Vars to detect statechanges on outputs 
	PreviousDim: BYTE;
	PreviousQ: BOOL;
	PreviousDBL: BOOL;
	/// Default values for dimmer, can be overwritten by method call 
	T_Debounce: TIME := TIME#10ms;
	T_Reconfig: TIME := TIME#10s0ms;
	T_On_Max: TIME := TIME#0ms;
	T_Dimm_Start: TIME := TIME#400ms;
	T_Dimm: TIME := TIME#3s0ms;
	Min_On: BYTE := 50;
	Max_On: BYTE := 255;
	Soft_Dimm: BOOL := TRUE;
	Dbl_Toggle: BOOL := FALSE;
	Rst_Out: BOOL := FALSE;
	/// Default value for click mode, can be overwritten by method call 
	T_Long: TIME := TIME#400ms;
END_VAR

FB_DIMMER(
	IN:= PB,
	SET:= SET,
	VAL:= VAL,
	RST:= RST,
	OUT:= DIM,
	T_DEBOUNCE:= T_Debounce,
	T_RECONFIG:= T_Reconfig,
	T_ON_MAX:= T_On_Max,
	T_DIMM_START:= T_Dimm_Start,
	T_DIMM:= T_Dimm,
	MIN_ON:= Min_On,
	MAX_ON:= Max_On,
	SOFT_DIMM:= Soft_Dimm,
	DBL_TOGGLE:= Dbl_Toggle,
	RST_OUT:= Rst_Out,
	Q=> Q,
	DBL=> DBL);
	
FB_DETECTPUSH(
	IN:= PB, 	
	SINGLE=> SINGLE, 
	DOUBLE=> DOUBLE, 
	TP_LONG=> LONG, 
	T_LONG:= T_long);
	
P_LONG_R_TRIG(CLK:=FB_DETECTPUSH.LONG);
P_LONG_F_TRIG(CLK:=FB_DETECTPUSH.LONG);
	
IF (ABS(BYTE_TO_INT(PreviousDim) - BYTE_TO_INT(DIM)) >= Delta_Dimm OR PB = FALSE) AND DIM <> PreviousDim AND OutputDimmer AND InitMqttDone  THEN
	PreviousDim:=DIM;
	pMqttPublishQueue^.AddMessage(		
		Payload := BYTE_TO_STRING(DIM),
		Topic := CONCAT(CONCAT(MqttPublishTopicPrefix^, MqttPublishTopicSuffix), '/DIM'),
		Qos := MQTT.QoS.ExactlyOnce,
		MqttRetain := FALSE
	);
END_IF

IF FB_DIMMER.Q <> PreviousQ AND InitMqttDone THEN
	PreviousQ:=FB_DIMMER.Q;
	pMqttPublishQueue^.AddMessage(
		Payload := BOOL_TO_STRING(FB_DIMMER.Q),
		Topic := CONCAT(CONCAT(MqttPublishTopicPrefix^, MqttPublishTopicSuffix), '/Q'),
		Qos := Qos_Dimm,
		MqttRetain := TRUE
	);
END_IF

IF FB_DIMMER.DBL <> PreviousDBL AND InitMqttDone THEN
	PreviousDBL:=FB_DIMMER.DBL;
	pMqttPublishQueue^.AddMessage(
		Payload := BOOL_TO_STRING(FB_DIMMER.DBL),
		Topic := CONCAT(CONCAT(MqttPublishTopicPrefix^, MqttPublishTopicSuffix), '/DBL'),
		Qos := MQTT.QoS.ExactlyOnce,
		MqttRetain := TRUE
	);
END_IF

IF FB_DETECTPUSH.SINGLE AND InitMqttDone THEN
	pMqttPublishQueue^.AddMessage(
		Payload := 'SINGLE',
		Topic := CONCAT(MqttPublishTopicPrefix^, MqttPublishTopicSuffix),
		Qos := MQTT.QoS.ExactlyOnce,
		MqttRetain := FALSE
	);
END_IF

IF FB_DETECTPUSH.DOUBLE AND InitMqttDone THEN
	pMqttPublishQueue^.AddMessage(
		Payload := 'DOUBLE',
		Topic := CONCAT(MqttPublishTopicPrefix^, MqttPublishTopicSuffix),
		Qos := MQTT.QoS.ExactlyOnce,
		MqttRetain := FALSE
	);
END_IF

IF FB_DETECTPUSH.TP_LONG AND InitMqttDone THEN
	pMqttPublishQueue^.AddMessage(
		Payload := 'LONG',
		Topic := CONCAT(MqttPublishTopicPrefix^, MqttPublishTopicSuffix),
		Qos := MQTT.QoS.ExactlyOnce,
		MqttRetain := FALSE
	);
END_IF

IF (P_LONG_R_TRIG.Q OR P_LONG_F_TRIG.Q) AND InitMqttDone THEN
	pMqttPublishQueue^.AddMessage(
		Payload := BOOL_TO_STRING(FB_DETECTPUSH.LONG),
		Topic := CONCAT(CONCAT(MqttPublishTopicPrefix^, MqttPublishTopicSuffix),'/P_LONG'),
		Qos := MQTT.QoS.ExactlyOnce,
		MqttRetain := TRUE
	);
END_IF

METHOD ConfigureFunctionBlock
VAR_INPUT
	/// Default values for dimmer, can be overwritten by method call 
	T_Debounce: TIME;
	T_Reconfig: TIME;
	T_On_Max: TIME;
	T_Dimm_Start: TIME;
	T_Dimm: TIME;
	Min_On: BYTE;
	Max_On: BYTE;
	Soft_Dimm: BOOL;
	Dbl_Toggle: BOOL;
	Rst_Out: BOOL;
	/// Default value for click mode, can be overwritten by method call 
	T_Long: TIME;
END_VAR
THIS^.T_Debounce:=T_Debounce;
THIS^.T_Reconfig:=T_Reconfig;
THIS^.T_On_Max:=T_On_Max;
THIS^.T_Dimm_Start:=T_Dimm_Start;
THIS^.T_Dimm:=T_Dimm;
THIS^.Min_On:=Min_On;
THIS^.Max_On:=Max_On;

THIS^.T_Long:=T_Long;
END_METHOD

METHOD InitMqtt
VAR_INPUT
	MQTTPublishPrefix: POINTER TO STRING;
	pMqttPublishQueue: POINTER TO FB_MqttPublishQueue;
	OutputDimmer: BOOL;
	Qos_Dimm: MQTT.QoS;
	Delta_Dimm: INT;
END_VAR
VAR
	InstanceNamePt: POINTER TO STRING;
END_VAR
THIS^.pMqttPublishQueue := pMqttPublishQueue;
THIS^.MqttPublishTopicPrefix := MQTTPublishPrefix;

InstanceNamePt := CommonTypesAndFunctions.FindLastDot(ADR(THIS^.InstanceName)) + 1;
THIS^.MqttPublishTopicSuffix := InstanceNamePt^;

THIS^.OutputDimmer:=OutputDimmer;
THIS^.Qos_Dimm:=Qos_Dimm;
THIS^.Delta_Dimm:=Delta_Dimm;

InitMqttDone := TRUE;
END_METHOD

END_FUNCTION_BLOCK

// FB_OUTPUT_BINARY_MQTT
{attribute 'reflection' := ''}
FUNCTION_BLOCK FB_OUTPUT_BINARY_MQTT EXTENDS FB_MQTT_BASE IMPLEMENTS MQTT.MQTT_SUBSCRIBE_CALLBACK
VAR_INPUT
	PRIO_HIGH: BOOL := FALSE;
	PRIO_LOW: BOOL := FALSE;
	TOGGLE: BOOL := FALSE;
END_VAR
VAR_OUTPUT
	OUT: BOOL;
END_VAR
VAR
	/// Refelection: object's full instance name
	{attribute 'noinit'}
	{attribute 'instance-path' := ''}
	InstancePath: STRING;
	Startup: BOOL := TRUE;
	///	ComposeJSONLight : STRUCT_TO_JSON;
	///	MqttDiscoveryMessageLight: MQTT_DISCOVERY_LIGHT;
	///	ComposeJSONLock : STRUCT_TO_JSON;
	///	MqttDiscoveryMessageLock: MQTT_DISCOVERY_LOCK;
	///	ComposeJSONSiren : STRUCT_TO_JSON;
	///	MqttDiscoveryMessageSiren: MQTT_DISCOVERY_SIREN;
	///	ComposeJSONSwitch : STRUCT_TO_JSON;
	///	
	MqttDiscMsgSwitch: MQTT_DISCOVERY_SWITCH;
END_VAR
VAR PERSISTENT
	/// To retain output state through powercycles
	PreviousState: BOOL;
END_VAR

IF Startup THEN
	OUT := PreviousState;
END_IF

IF PRIO_HIGH THEN
	OUT:=TRUE;
ELSIF(PRIO_LOW AND NOT (PRIO_HIGH)) THEN
	OUT:= FALSE;
ELSIF MqttHighRequest THEN
	OUT:= TRUE;
	MqttHighRequest := FALSE;
	MqttLowRequest := FALSE;
ELSIF MqttLowRequest THEN
	OUT:= FALSE;
	MqttHighRequest := FALSE;
	MqttLowRequest := FALSE;
ELSIF(TOGGLE) THEN
	OUT:=NOT(OUT);
END_IF;

IF ((PreviousState <> OUT) OR Startup) AND InitMqttDone THEN
	pMqttPublishQueue^.AddMessage(
		Payload := BOOL_TO_STRING(OUT),
		Topic := MQTTPublishTopic,
		Qos := MQTT.QoS.ExactlyOnce,
		MqttRetain := TRUE
	);	
	Startup:=FALSE;
END_IF	

PreviousState := OUT;

METHOD InitMqtt
VAR_INPUT
	MQTTPublishPrefix: POINTER TO STRING;
	MQTTSubscribePrefix: POINTER TO STRING;
	pMqttPublishQueue: POINTER TO FB_MqttPublishQueue;
	pMqttCallbackCollector: POINTER TO MQTT.CallbackCollector;
END_VAR
SUPER^._InstancePath := THIS^.InstancePath; // Due to reflection its location is important

(*pass trough*)
THIS^.pMqttPublishQueue := pMqttPublishQueue;
THIS^.MqttPublishTopicPrefix:=MQTTPublishPrefix;
THIS^.MQTTSubscribeTopicPrefix:=MQTTSubscribePrefix;
THIS^.pMqttPublishQueue:=pMqttPublishQueue;

SUPER^.InitBaseMqtt();
pMqttCallbackCollector^.put(instance:= THIS^); // register the FB agains the collector so mqtt events can be received
END_METHOD

METHOD InitMqttDiscoveryAsLight
VAR_INPUT
	Device: POINTER TO FB_PLC_MQTT_DISCOVERY_DEVICE;
	Name: STRING(255);
	overruleId: STRING(255) := '';
	meta: STRING(255) := '';
	Invert: BOOL := FALSE;
END_VAR
VAR
	id: STRING(255);
END_VAR
IF InitMqttDone AND NOT initMqttDiscoveryDone THEN
	
	IF CommonTypesAndFunctions.StrEquals(str1:= ADR(overruleId), str2:= ADR('')) THEN
		id := CONCAT(CONCAT(THIS^.DeviceName,'_'), THIS^.InstanceNamePt^); // 'FB_DI_PB_003'
	ELSE
		id := overruleId; // 'MY_PH_GND_HALL_01'
	END_IF
	
	Device^.CreateLightEntity(
			Name := name,
			Id := id,
			Meta := meta,
			CommandTopic := THIS^.MQTTSubscribeTopic,
			PayloadOn := BOOL_TO_STRING(NOT(Invert)),
			PayloadOff := BOOL_TO_STRING(Invert),
			StateTopic := THIS^.MQTTPublishTopic);

	initMqttDiscoveryDone := TRUE;
END_IF
END_METHOD

METHOD InitMqttDiscoveryAsLock
VAR_INPUT
	Device: POINTER TO FB_PLC_MQTT_DISCOVERY_DEVICE;
	Name: STRING(255);
	overruleId: STRING(255) := '';
	meta: STRING(255) := '';
	Invert: BOOL := FALSE;
END_VAR
VAR
	id: STRING(255);
END_VAR
IF InitMqttDone AND NOT initMqttDiscoveryDone THEN
	
	IF CommonTypesAndFunctions.StrEquals(str1:= ADR(overruleId), str2:= ADR('')) THEN
		id := CONCAT(CONCAT(THIS^.DeviceName,'_'), THIS^.InstanceNamePt^); // 'FB_DI_PB_003'
	ELSE
		id := overruleId; // 'MY_PH_GND_HALL_01'
	END_IF
	
	Device^.CreateLockEntity(
		Name := name,
		Id := id,
		Meta := meta,
		CommandTopic := THIS^.MQTTSubscribeTopic,
		PayloadLock := BOOL_TO_STRING(NOT(Invert)),
		PayloadUnlock := BOOL_TO_STRING(Invert),
		StateTopic := THIS^.MQTTPublishTopic,
		StateUnlocked := BOOL_TO_STRING(Invert),
		StateLocked := BOOL_TO_STRING(NOT(Invert)));

	initMqttDiscoveryDone := TRUE;
END_IF
END_METHOD

METHOD InitMqttDiscoveryAsSiren
VAR_INPUT
	Device: POINTER TO FB_PLC_MQTT_DISCOVERY_DEVICE;
	Name: STRING(255);
	overruleId: STRING(255) := '';
	meta: STRING(255) := '';
	Invert: BOOL := FALSE;
END_VAR
VAR
	id: STRING(255);
END_VAR
IF InitMqttDone AND NOT initMqttDiscoveryDone THEN
	
	IF CommonTypesAndFunctions.StrEquals(str1:= ADR(overruleId), str2:= ADR('')) THEN
		id := CONCAT(CONCAT(THIS^.DeviceName,'_'), THIS^.InstanceNamePt^); // 'FB_DI_PB_003'
	ELSE
		id := overruleId; // 'MY_PH_GND_HALL_01'
	END_IF
	
	Device^.CreateSirenEntity(
			Name := name,
			Id := id,
			Meta := meta,
			CommandTopic := THIS^.MQTTSubscribeTopic,
			PayloadOn := BOOL_TO_STRING(NOT(Invert)),
			PayloadOff := BOOL_TO_STRING(Invert),
			StateTopic := THIS^.MQTTPublishTopic,
			StateOnPayload := BOOL_TO_STRING(NOT(Invert)),
			StateOffPayload := BOOL_TO_STRING(Invert)
		);


	initMqttDiscoveryDone := TRUE;
END_IF
END_METHOD

METHOD InitMqttDiscoveryAsSwitch
VAR_INPUT
	Device: POINTER TO FB_PLC_MQTT_DISCOVERY_DEVICE;
	Name: STRING(255);
	DeviceClass: STRING(100) := 'outlet';
	overruleId: STRING(255) := '';
	meta: STRING(255) := '';
	Invert: BOOL := FALSE;
END_VAR
VAR
	id: STRING(255);
END_VAR
IF InitMqttDone AND NOT initMqttDiscoveryDone THEN
	
	IF CommonTypesAndFunctions.StrEquals(str1:= ADR(overruleId), str2:= ADR('')) THEN
		id := CONCAT(CONCAT(THIS^.DeviceName,'_'), THIS^.InstanceNamePt^); // 'FB_DI_PB_003'
	ELSE
		id := overruleId; // 'MY_PH_GND_HALL_01'
	END_IF
	
	Device^.CreateSwitchEntity(
			Name := name,
			Id := id,
			Meta := meta,
			CommandTopic := THIS^.MQTTSubscribeTopic,
			PayloadOn := BOOL_TO_STRING(NOT(Invert)),
			PayloadOff := BOOL_TO_STRING(Invert),
			StateTopic := THIS^.MQTTPublishTopic,
			StateOnPayload := BOOL_TO_STRING(NOT(Invert)),
			StateOffPayload := BOOL_TO_STRING(Invert),
			DeviceClass := DeviceClass);
	
	initMqttDiscoveryDone := TRUE;
END_IF
END_METHOD

METHOD PublishReceived : BOOL
VAR_INPUT
	///Collection of recived Data
	Data: MQTT.CALLBACK_DATA;
END_VAR
//first check if Mqtt is initialized, otherwise do nothing
IF NOT(InitMqttDone) THEN
	//mark the interface call from the collector as done
	PublishReceived := TRUE;
//check if the packet is for this FB
ELSIF CommonTypesAndFunctions.StrEquals(str1:= ADR(MQTTSubscribeTopic), str2:= Data.TopicOut) THEN
	//mark the interface call from the collector as done
	PublishReceived := TRUE;
	//now process the data
	IF CommonTypesAndFunctions.StrEquals(str1:= Data.PayloadString, str2:= ADR('TRUE')) THEN
		MqttHighRequest := TRUE;
	ELSIF CommonTypesAndFunctions.StrEquals(str1:= Data.PayloadString, str2:= ADR('FALSE')) THEN
		MqttLowRequest := TRUE;
	// Siren sends out a JSON
	ELSIF FIND(Data.PayloadString^, 'TRUE') > 0 THEN
		MqttHighRequest := TRUE;
	ELSIF FIND(Data.PayloadString^, 'FALSE') > 0 THEN
		MqttLowRequest := TRUE;
	END_IF
END_IF
END_METHOD

END_FUNCTION_BLOCK

// FB_OUTPUT_BISTABLE_MQTT
{attribute 'reflection' := ''}
FUNCTION_BLOCK FB_OUTPUT_BISTABLE_MQTT EXTENDS FB_MQTT_BASE IMPLEMENTS MQTT.MQTT_SUBSCRIBE_CALLBACK
VAR_INPUT
	PRIO_HIGH: BOOL := FALSE;
	PRIO_LOW: BOOL := FALSE;
	TOGGLE: BOOL := FALSE;
	FEEDBACK: BOOL := FALSE;
END_VAR
VAR_OUTPUT
	OUT: BOOL;
END_VAR
VAR
	/// Refelection: object's full instance name
	{attribute 'noinit'}
	{attribute 'instance-path' := ''}
	InstancePath: STRING;
	Startup: BOOL := TRUE;
	PreviousFeedback: BOOL;
	HoldTimer: TOF;
	T_hold: TIME := TIME#1s0ms;
	PulseTrigger: BOOL := FALSE;
	MqttDiscoveryMessageLight: MQTT_DISCOVERY_LIGHT;
	MqttDiscoveryMessageLock: MQTT_DISCOVERY_LOCK;
	MqttDiscoveryMessageSiren: MQTT_DISCOVERY_SIREN;
	MqttDiscoveryMessageSwitch: MQTT_DISCOVERY_SWITCH;
END_VAR

HoldTimer(PT:= T_hold);

IF PRIO_HIGH THEN
	IF NOT FEEDBACK THEN
		PulseTrigger:=TRUE;
	END_IF
ELSIF(PRIO_LOW AND NOT (PRIO_HIGH)) THEN
	IF FEEDBACK THEN		
		PulseTrigger:=TRUE;
	END_IF
	OUT:= FALSE;
ELSIF MqttHighRequest THEN
	IF NOT FEEDBACK THEN		
		PulseTrigger:=TRUE;
	END_IF
	MqttHighRequest := FALSE;
	MqttLowRequest := FALSE;
ELSIF MqttLowRequest THEN
	IF FEEDBACK THEN		
		PulseTrigger:=TRUE;
	END_IF
	MqttHighRequest := FALSE;
	MqttLowRequest := FALSE;
ELSIF(TOGGLE) THEN	
	PulseTrigger:=TRUE;
END_IF;

IF ((PreviousFeedback <> FEEDBACK) OR Startup) AND InitMqttDone THEN
	pMqttPublishQueue^.AddMessage(
		Payload := BOOL_TO_STRING(FEEDBACK),
		Topic := CONCAT(MqttPublishTopicPrefix^, MqttPublishTopicSuffix),
		Qos := MQTT.QoS.ExactlyOnce,
		MqttRetain := TRUE
	);	
	Startup:=FALSE;
END_IF	

PreviousFeedback := FEEDBACK;
HoldTimer.IN	 := PulseTrigger;
OUT := HoldTimer.Q;

PulseTrigger:=FALSE;

METHOD ConfigureFunctionBlock
VAR_INPUT
	/// Default value for click mode, can be overwritten by method call 
	T_hold: TIME;
END_VAR
THIS^.T_hold:=T_hold;
END_METHOD

METHOD InitMqtt
VAR_INPUT
	MQTTPublishPrefix: POINTER TO STRING;
	MQTTSubscribePrefix: POINTER TO STRING;
	pMqttPublishQueue: POINTER TO FB_MqttPublishQueue;
	pMqttCallbackCollector: POINTER TO MQTT.CallbackCollector;
END_VAR
SUPER^._InstancePath := THIS^.InstancePath; // Due to reflection its location is important

(*pass trough*)
THIS^.pMqttPublishQueue := pMqttPublishQueue;
THIS^.MqttPublishTopicPrefix:=MQTTPublishPrefix;
THIS^.MQTTSubscribeTopicPrefix:=MQTTSubscribePrefix;
THIS^.pMqttPublishQueue:=pMqttPublishQueue;



SUPER^.InitBaseMqtt();
pMqttCallbackCollector^.put(instance:= THIS^); // register the FB agains the collector so mqtt events can be received
END_METHOD

METHOD InitMqttDiscoveryAsLight
VAR_INPUT
	Device: POINTER TO FB_PLC_MQTT_DISCOVERY_DEVICE;
	Name: STRING(255);
	overruleId: STRING(255) := '';
	meta: STRING(255) := '';
	Invert: BOOL := FALSE;
END_VAR
VAR
	id: STRING(255);
END_VAR
IF InitMqttDone AND NOT initMqttDiscoveryDone THEN
	
	IF CommonTypesAndFunctions.StrEquals(str1:= ADR(overruleId), str2:= ADR('')) THEN
		id := CONCAT(CONCAT(THIS^.DeviceName,'_'), THIS^.InstanceNamePt^); // 'FB_DI_PB_003'
	ELSE
		id := overruleId; // 'MY_PH_GND_HALL_01'
	END_IF
	
	Device^.CreateLightEntity(
			Name := name,
			Id := id,
			Meta := meta,
			CommandTopic := THIS^.MQTTSubscribeTopic,
			PayloadOn := BOOL_TO_STRING(NOT(Invert)),
			PayloadOff := BOOL_TO_STRING(Invert),
			StateTopic := THIS^.MQTTPublishTopic);

	initMqttDiscoveryDone := TRUE;
END_IF
END_METHOD

METHOD InitMqttDiscoveryAsLock
VAR_INPUT
	Device: POINTER TO FB_PLC_MQTT_DISCOVERY_DEVICE;
	Name: STRING(255);
	overruleId: STRING(255) := '';
	meta: STRING(255) := '';
	Invert: BOOL := FALSE;
END_VAR
VAR
	id: STRING(255);
END_VAR
IF InitMqttDone AND NOT initMqttDiscoveryDone THEN
	
	IF CommonTypesAndFunctions.StrEquals(str1:= ADR(overruleId), str2:= ADR('')) THEN
		id := CONCAT(CONCAT(THIS^.DeviceName,'_'), THIS^.InstanceNamePt^); // 'FB_DI_PB_003'
	ELSE
		id := overruleId; // 'MY_PH_GND_HALL_01'
	END_IF
	
	Device^.CreateLockEntity(
		Name := name,
		Id := id,
		Meta := meta,
		CommandTopic := THIS^.MQTTSubscribeTopic,
		PayloadLock := BOOL_TO_STRING(NOT(Invert)),
		PayloadUnlock := BOOL_TO_STRING(Invert),
		StateTopic := THIS^.MQTTPublishTopic,
		StateUnlocked := BOOL_TO_STRING(Invert),
		StateLocked := BOOL_TO_STRING(NOT(Invert)));

	initMqttDiscoveryDone := TRUE;
END_IF
END_METHOD

METHOD InitMqttDiscoveryAsSiren
VAR_INPUT
	Device: POINTER TO FB_PLC_MQTT_DISCOVERY_DEVICE;
	Name: STRING(255);
	overruleId: STRING(255) := '';
	meta: STRING(255) := '';
	Invert: BOOL := FALSE;
END_VAR
VAR
	id: STRING(255);
END_VAR
IF InitMqttDone AND NOT initMqttDiscoveryDone THEN
	
	IF CommonTypesAndFunctions.StrEquals(str1:= ADR(overruleId), str2:= ADR('')) THEN
		id := CONCAT(CONCAT(THIS^.DeviceName,'_'), THIS^.InstanceNamePt^); // 'FB_DI_PB_003'
	ELSE
		id := overruleId; // 'MY_PH_GND_HALL_01'
	END_IF
	
	Device^.CreateSirenEntity(
			Name := name,
			Id := id,
			Meta := meta,
			CommandTopic := THIS^.MQTTSubscribeTopic,
			PayloadOn := BOOL_TO_STRING(NOT(Invert)),
			PayloadOff := BOOL_TO_STRING(Invert),
			StateTopic := THIS^.MQTTPublishTopic,
			StateOnPayload := BOOL_TO_STRING(NOT(Invert)),
			StateOffPayload := BOOL_TO_STRING(Invert)
		);

	initMqttDiscoveryDone := TRUE;
END_IF
END_METHOD

METHOD InitMqttDiscoveryAsSwitch
VAR_INPUT
	Device: POINTER TO FB_PLC_MQTT_DISCOVERY_DEVICE;
	Name: STRING(255);
	DeviceClass: STRING(100) := 'outlet';
	overruleId: STRING(255) := '';
	meta: STRING(255) := '';
	Invert: BOOL := FALSE;
END_VAR
VAR
	id: STRING(255);
END_VAR
IF InitMqttDone AND NOT initMqttDiscoveryDone THEN
	
	IF CommonTypesAndFunctions.StrEquals(str1:= ADR(overruleId), str2:= ADR('')) THEN
		id := CONCAT(CONCAT(THIS^.DeviceName,'_'), THIS^.InstanceNamePt^); // 'FB_DI_PB_003'
	ELSE
		id := overruleId; // 'MY_PH_GND_HALL_01'
	END_IF
	
	Device^.CreateSwitchEntity(
			Name := name,
			Id := id,
			Meta := meta,
			CommandTopic := THIS^.MQTTSubscribeTopic,
			PayloadOn := BOOL_TO_STRING(NOT(Invert)),
			PayloadOff := BOOL_TO_STRING(Invert),
			StateTopic := THIS^.MQTTPublishTopic,
			StateOnPayload := BOOL_TO_STRING(NOT(Invert)),
			StateOffPayload := BOOL_TO_STRING(Invert),
			DeviceClass := DeviceClass);
	
	initMqttDiscoveryDone := TRUE;
END_IF
END_METHOD

METHOD PublishReceived : BOOL
VAR_INPUT
	///Collection of recived Data
	Data: MQTT.CALLBACK_DATA;
END_VAR
//first check if Mqtt is initialized, otherwise do nothing
IF NOT(InitMqttDone) THEN
	//mark the interface call from the collector as done
	PublishReceived := TRUE;
//check if the packet is for this FB
ELSIF CommonTypesAndFunctions.StrEquals(str1:= ADR(MQTTSubscribeTopic), str2:= Data.TopicOut) THEN
	//mark the interface call from the collector as done
	PublishReceived := TRUE;
	//now process the data
	IF CommonTypesAndFunctions.StrEquals(str1:= Data.PayloadString, str2:= ADR('TRUE')) THEN
		MqttHighRequest := TRUE;
	ELSIF CommonTypesAndFunctions.StrEquals(str1:= Data.PayloadString, str2:= ADR('FALSE')) THEN
		MqttLowRequest := TRUE;
	// Siren sends out a JSON
	ELSIF FIND(Data.PayloadString^, 'TRUE') > 0 THEN
		MqttHighRequest := TRUE;
	ELSIF FIND(Data.PayloadString^, 'FALSE') > 0 THEN
		MqttLowRequest := TRUE;
	END_IF
END_IF
END_METHOD

END_FUNCTION_BLOCK

// FB_OUTPUT_COVER_MQTT
{attribute 'reflection' := ''}
FUNCTION_BLOCK FB_OUTPUT_COVER_MQTT EXTENDS FB_MQTT_BASE IMPLEMENTS MQTT.MQTT_SUBSCRIBE_CALLBACK
VAR_INPUT
	TOGGLE: BOOL;
	PRIO_LOCK: BOOL;
	PRIO_UP: BOOL;
	PRIO_DN: BOOL;
	{attribute 'input_constant' := ''}
	T_LOCKOUT: TIME := TIME#1s0ms;
	{attribute 'input_constant' := ''}
	T_UD: TIME := TIME#10s0ms;
END_VAR
VAR_OUTPUT
	MU: BOOL;
	MD: BOOL;
END_VAR
VAR
	/// object's full instance name 
	{attribute 'instance-path' := ''}
	{attribute 'noinit'}
	InstancePath: STRING;
	lock: OSCAT_BASIC.INTERLOCK;
	Cover_State_Timer: TOF;
	internalUp: BOOL;
	internalDown: BOOL;
	MqttRequestStop: BOOL;
	MqttRequestOpen: BOOL;
	MqttRequestClose: BOOL;
	MqttDiscoveryMessage: MQTT_DISCOVERY_COVER;
END_VAR
VAR PERSISTENT
	///down = false, up = true
	internalDir: BOOL;
END_VAR

(* Run the timer to not power the motors for to long *)
Cover_State_Timer(PT:=T_UD);
Cover_State_Timer.IN:=FALSE;

IF NOT(Cover_State_Timer.Q) AND internalUp THEN
	pMqttPublishQueue^.AddMessage(
		Payload := 'OPEN',
		Topic := CONCAT(MqttPublishTopicPrefix^, MqttPublishTopicSuffix),
		Qos := MQTT.QoS.ExactlyOnce,
		MqttRetain := TRUE
	);
END_IF

IF NOT(Cover_State_Timer.Q) AND internalDown THEN
	pMqttPublishQueue^.AddMessage(
		Payload := 'CLOSED',
		Topic := CONCAT(MqttPublishTopicPrefix^, MqttPublishTopicSuffix),
		Qos := MQTT.QoS.ExactlyOnce,
		MqttRetain := TRUE
	);
END_IF


(* Check what to do *)
IF NOT(Cover_State_Timer.Q) AND internalUp THEN // don't run the motors for to long, assume we've reached end and toggle dir
	internalUp := FALSE;
	internalDown := FALSE;
	internalDir := FALSE;
ELSIF NOT(Cover_State_Timer.Q) AND internalDown THEN // don't run the motors for to long, assume we've reached end and toggle dir
	internalUp := FALSE;
	internalDown := FALSE;
	internalDir := TRUE;
ELSIF PRIO_LOCK THEN	
	internalUp := FALSE;
	internalDown := FALSE;
ELSIF PRIO_UP THEN	
	internalUp := TRUE;
	internalDown := FALSE;
	Cover_State_Timer.IN:=TRUE;
ELSIF PRIO_DN THEN	
	internalUp := FALSE;
	internalDown := TRUE;
	Cover_State_Timer.IN:=TRUE;
ELSIF TOGGLE AND (internalUp OR internalDown) THEN	// stop and toggle dir
	internalUp := FALSE;
	internalDown := FALSE;
	internalDir := NOT(internalDir);
ELSIF TOGGLE AND NOT(internalDir) THEN //move down
	internalUp := FALSE;
	internalDown := TRUE;
	Cover_State_Timer.IN:=TRUE;
ELSIF TOGGLE AND internalDir THEN //move upwards
	internalUp := TRUE;
	internalDown := FALSE;	
	Cover_State_Timer.IN:=TRUE;
ELSIF MqttRequestStop THEN
	internalUp := FALSE;
	internalDown := FALSE;
	MqttRequestStop := FALSE;
ELSIF MqttRequestOpen THEN
	internalUp := TRUE;
	internalDown := FALSE;
	MqttRequestOpen := FALSE;
	Cover_State_Timer.IN:=TRUE;;
ELSIF MqttRequestClose THEN
	internalUp := FALSE;
	internalDown := TRUE;
	MqttRequestClose := FALSE;
	Cover_State_Timer.IN:=TRUE;
END_IF

(* make sure only one motor is active at a given time *)
lock(i1 := internalUp, I2 := InternalDown, TL := T_lockout);
MU := lock.Q1;
MD := lock.Q2;

METHOD ConfigureFunctionBlock : BOOL
VAR_INPUT
	T_LOCKOUT: TIME;
	T_UD: TIME;
END_VAR
THIS^.T_LOCKOUT:=T_LOCKOUT;
THIS^.T_UD:=T_UD;
END_METHOD

METHOD InitMqtt
VAR_INPUT
	MQTTPublishPrefix: POINTER TO STRING;
	MQTTSubscribePrefix: POINTER TO STRING;
	pMqttPublishQueue: POINTER TO FB_MqttPublishQueue;
	pMqttCallbackCollector: POINTER TO MQTT.CallbackCollector;
END_VAR
VAR
	InstanceNamePt: POINTER TO STRING;
END_VAR
SUPER^._InstancePath := THIS^.InstancePath; // Due to reflection its location is important

(*pass trough*)
THIS^.pMqttPublishQueue := pMqttPublishQueue;
THIS^.MqttPublishTopicPrefix:=MQTTPublishPrefix;
THIS^.MQTTSubscribeTopicPrefix:=MQTTSubscribePrefix;
THIS^.pMqttPublishQueue:=pMqttPublishQueue;

SUPER^.InitBaseMqtt();
pMqttCallbackCollector^.put(instance:= THIS^); // register the FB agains the collector so mqtt events can be received
END_METHOD

METHOD InitMqttDiscovery
VAR_INPUT
	Device: POINTER TO FB_PLC_MQTT_DISCOVERY_DEVICE;
	Name: STRING(255);
	overruleId: STRING(255) := '';
	meta: STRING(255) := '';
	DeviceClass: STRING(50) := 'shutter';
END_VAR
VAR
	id: STRING(255);
END_VAR
IF InitMqttDone AND NOT initMqttDiscoveryDone THEN
	
	IF CommonTypesAndFunctions.StrEquals(str1:= ADR(overruleId), str2:= ADR('')) THEN
		id := CONCAT(CONCAT(THIS^.DeviceName,'_'), THIS^.InstanceNamePt^); // 'FB_DI_PB_003'
	ELSE
		id := overruleId; // 'MY_PH_GND_HALL_01'
	END_IF
	
	Device^.CreateCoverEntity(
		Name := name,
		Id := id,
		Meta := meta,
		CommandTopic := THIS^.MQTTSubscribeTopic,
		PayloadOpen := 'OPEN',
		PayloadClose := 'CLOSE',
		PayloadStop := 'STOP',
		StateTopic := THIS^.MQTTPublishTopic,
		StateOpen := 'OPEN',
		StateClosed := 'CLOSED',
		DeviceClass := DeviceClass
	);

	initMqttDiscoveryDone := TRUE;
END_IF
END_METHOD

METHOD PublishReceived : BOOL
VAR_INPUT
	///Collection of recived Data
	Data: MQTT.CALLBACK_DATA;
END_VAR
//first check if Mqtt is initialized, otherwise do nothing
IF NOT(InitMqttDone) THEN
	//mark the interface call from the collector as done
	PublishReceived := TRUE;
//check if the packet is for this FB
ELSIF CommonTypesAndFunctions.StrEquals(str1:= ADR(MQTTSubscribeTopic), str2:= Data.TopicOut) THEN
	//mark the interface call from the collector as done
	PublishReceived := TRUE;
	//now process the data
	IF CommonTypesAndFunctions.StrEquals(str1:= Data.PayloadString, str2:= ADR('STOP')) THEN			
		THIS^.MqttRequestStop:=TRUE;
	ELSIF CommonTypesAndFunctions.StrEquals(str1:= Data.PayloadString, str2:= ADR('OPEN')) THEN
		THIS^.MqttRequestOpen:=TRUE;
	ELSIF CommonTypesAndFunctions.StrEquals(str1:= Data.PayloadString, str2:= ADR('CLOSE')) THEN
		THIS^.MqttRequestClose:=TRUE;
	END_IF

END_IF
END_METHOD

END_FUNCTION_BLOCK

// FB_OUTPUT_DIMMER_MQTT
{attribute 'reflection' := ''}
FUNCTION_BLOCK FB_OUTPUT_DIMMER_MQTT EXTENDS FB_MQTT_BASE IMPLEMENTS MQTT.MQTT_SUBSCRIBE_CALLBACK
VAR_INPUT
	SINGLE: BOOL;
	LONG: BOOL;
	P_LONG: BOOL;
	PRIO_HIGH: BOOL := FALSE;
	PRIO_LOW: BOOL := FALSE;
	SET: BOOL;
	VAL: BYTE;
	RST: BOOL;
END_VAR
VAR_OUTPUT
	Q: BOOL;
	Q_OUT: WORD;
	OUT: WORD;
END_VAR
VAR
	/// Refelection: object's full instance name
	{attribute 'instance-path' := ''}
	{attribute 'noinit'}
	InstancePath: STRING;
	t3: OSCAT_BASIC.TON;
	dim: OSCAT_BASIC._RMP_B;
	dir: BOOL;
	OUT_Internal: BYTE;
	LIN_TRAFO: Util.LIN_TRAFO;
	enabled: BOOL := TRUE;
	Startup: BOOL := TRUE;
	OutputDimmer: BOOL;
	Qos_Dimm: MQTT.QoS;
	Delta_Dimm: INT;
	/// Default values for dimmer, can be overwritten by method call 
	T_Debounce: TIME := TIME#10ms;
	T_Reconfig: TIME := TIME#10s0ms;
	T_On_Max: TIME := TIME#0ms;
	T_Dimm_Start: TIME := TIME#400ms;
	T_Dimm: TIME := TIME#1s0ms;
	Min_On: BYTE := 100;
	Max_On: BYTE := 200;
	Soft_Dimm: BOOL := TRUE;
	Rst_Out: BOOL := FALSE;
	OUT_LinearScaleMin: INT := 10000;
	OUT_LinearScaleMax: INT := 32767;
	/// DMX specific 
	DmxChannel: INT;
	DmxWidth: INT;
	DmxUniverse: INT;
	pDmxValues: POINTER TO oscat_network.NETWORK_BUFFER_SHORT;
	InitDmxDone: BOOL := FALSE;
	OUT_Target: BYTE;
	SoftDimToValue: BOOL;
	SoftDimToQFalse: BOOL;
	UpdateValueStep: BYTE := 4;
	OUT_Internal_tmp: BYTE;
	curve: DINT := DIMMER_CURVE.linear;
	wait: TON;
	Step: INT := 0;
	dimmedValue: INT := 1;
	/// one time before and after blink
	waitTimeAtTop: TIME := TIME#200ms;
	blinkValue: BYTE := 100;
	blinkEnabled: BOOL := FALSE;
	MqttDiscoveryMessage: MQTT_DISCOVERY_LIGHT_DIMMER;
END_VAR
VAR PERSISTENT
	/// To retain output state through powercycles
	PreviousOUT: BYTE;
	/// To retain output state through powercycles
	PreviousQ: BOOL;
END_VAR



IF Startup THEN
	OUT := PreviousOUT;
	Q := PreviousQ;
END_IF

IF RST THEN
	IF rst_out THEN OUT_Internal := 0; END_IF;
	Q := FALSE;
	dir := OUT_Internal > 127;
ELSIF PRIO_HIGH THEN
	Q := TRUE;
	OUT_Internal := 255;
ELSIF PRIO_LOW THEN
	Q := FALSE;
ELSIF MqttHighRequest THEN
	Q:= TRUE;
	MqttHighRequest := FALSE;
	MqttLowRequest := FALSE;
ELSIF MqttLowRequest THEN
	Q:= FALSE;
	MqttHighRequest := FALSE;
	MqttLowRequest := FALSE;
ELSIF set THEN
	OUT_Internal := val;
	Q := TRUE;
	(* set direction to up when value < 127 otherwise set dir down dir is reversed because next action will reverse again *)
	dir := OUT_Internal > 127;
ELSIF SINGLE THEN
	(* a single click reverses output Q *)
	Q := NOT Q;
	(* when dimmer is turned on we need to limit out to min and max limits *)
	IF Q THEN OUT_Internal := LIMIT(MAX(OUT_Internal,1), OUT_Internal, MAX_ON);	END_IF;
	(* set the appropriate direction of dimmer dir is reversed because next action will reverse again *)
	dir := OUT_Internal > 127;
ELSIF LONG THEN
	IF NOT Q THEN
		IF SOFT_DIMM THEN
			OUT_Internal := 1;
			dir := TRUE;
		ELSE
			OUT_Internal := LIMIT(MAX(MIN_ON,1), OUT_Internal, MAX_ON);
			DIR := OUT_Internal < 127;
		END_IF;
		Q := TRUE;
	ELSE
		(* reverse direction with every long click *)
		dir := NOT dir;
	END_IF;
END_IF;


(* while dimming is active ramp the output out up or down *)
dim(DIR := dir, e := P_LONG AND Q, TR := T_DIMM, rmp := OUT_Internal);

(* reverse direction when limits are reached *)
IF OUT_Internal = 0 THEN
	dir := TRUE;
ELSIF OUT_Internal = 255 THEN
	dir := FALSE;
END_IF;

(* limit the maximum runtime *)
IF t_ON_MAX > t#0s THEN
	t3(in := q, pt := T_ON_MAX);
	Q := Q XOR t3.Q;
END_IF;

(* Scale the internal OUT to the actual OUT *)
LIN_TRAFO(
		IN:= OUT_Internal,
		IN_MIN:= 0,
		IN_MAX:= 255,
		OUT_MIN:=OUT_LinearScaleMin,
		OUT_MAX:=OUT_LinearScaleMax
	);
OUT:= REAL_TO_WORD(LIN_TRAFO.OUT);
IF Q THEN
	Q_OUT:= OUT;
ELSE
	Q_OUT:= 0;
END_IF

IF ((ABS(BYTE_TO_INT(PreviousOUT) - BYTE_TO_INT(OUT_Internal)) >= Delta_Dimm) OR Startup AND OUT_Internal <> PreviousOUT OR Startup AND OutputDimmer) AND InitMqttDone THEN
	PreviousOUT:=OUT_Internal;
	pMqttPublishQueue^.AddMessage(		
		Payload := BYTE_TO_STRING(OUT_Internal),
		Topic := CONCAT(THIS^.MQTTPublishTopic,'/OUT'),
		Qos := MQTT.QoS.ExactlyOnce,
		MqttRetain := TRUE
	);
END_IF

IF (Q <> PreviousQ OR Startup) AND InitMqttDone THEN
	PreviousQ:=Q;
	pMqttPublishQueue^.AddMessage(
		Payload := BOOL_TO_STRING(Q),
		Topic := CONCAT(THIS^.MQTTPublishTopic,'/Q'),
		Qos := Qos_Dimm,
		MqttRetain := TRUE
	);
END_IF

Startup:=FALSE;

(* DMX specific *)
IF InitDmxDone THEN 
	IF Q THEN
		IF pDmxValues^.BUFFER[DmxChannel-1] <> OUT_Internal THEN
			pDmxValues^.BUFFER[DmxChannel-1] := OUT_Internal;
		END_IF
	ELSE 
		IF pDmxValues^.BUFFER[DmxChannel-1] <> 0 THEN
			pDmxValues^.BUFFER[DmxChannel-1] := 0;
		END_IF
	END_IF
END_IF
IF SoftDimToValue AND OUT_Internal = OUT_Target THEN // If the same, softdim to value is done
	SoftDimToValue := FALSE;
	IF SoftDimToQFalse THEN
		SoftDimToQFalse := FALSE;
		OUT_Internal := OUT_Internal_tmp;
		PreviousOUT:=OUT_Internal;
	END_IF
END_IF
Startup:=FALSE;

(* DMX specific *)

METHOD ConfigureFunctionBlock
VAR_INPUT
	/// Default values for dimmer, can be overwritten by method call 
	T_Debounce: TIME := TIME#10ms;
	T_Reconfig: TIME := TIME#10s0ms;
	T_On_Max: TIME := TIME#0ms;
	T_Dimm_Start: TIME := TIME#400ms;
	T_Dimm: TIME := TIME#3s0ms;
	Min_On: BYTE := 50;
	Max_On: BYTE := 255;
	Soft_Dimm: BOOL := TRUE;
	Rst_Out: BOOL := FALSE;
	OUT_LinearScaleMin: INT := 0;
	OUT_LinearScaleMax: INT := 32767;
END_VAR
THIS^.T_Debounce:=T_Debounce;
THIS^.T_Reconfig:=T_Reconfig;
THIS^.T_On_Max:=T_On_Max;
THIS^.T_Dimm_Start:=T_Dimm_Start;
THIS^.T_Dimm:=T_Dimm;
THIS^.Min_On:=Min_On;
THIS^.Max_On:=Max_On;
THIS^.Soft_Dimm:=Soft_Dimm;
THIS^.Rst_Out:=Rst_Out;
THIS^.OUT_LinearScaleMin:=OUT_LinearScaleMin;
THIS^.OUT_LinearScaleMax:=OUT_LinearScaleMax;
END_METHOD

METHOD initDMX
VAR_INPUT
	DmxChannel: INT;
	DmxWidth: INT := 1;
	DmxUniverse: INT := 1;
	pDmxValues: POINTER TO oscat_network.NETWORK_BUFFER_SHORT;
END_VAR

IF NOT THIS^.InitDmxDone THEN
	THIS^.DmxChannel := DmxChannel;
	THIS^.pDmxValues := pDmxValues;
	THIS^.DmxWidth := DmxWidth;
	THIS^.InitDmxDone := TRUE;
	
	THIS^.InitDmxDone := TRUE;
END_IF
END_METHOD

METHOD InitMqtt
VAR_INPUT
	MQTTPublishPrefix: POINTER TO STRING;
	MQTTSubscribePrefix: POINTER TO STRING;
	pMqttPublishQueue: POINTER TO FB_MqttPublishQueue;
	pMqttCallbackCollector: POINTER TO MQTT.CallbackCollector;
	/// Dimmer specific
	OutputDimmer: BOOL;
	Qos_Dimm: MQTT.QoS;
	Delta_Dimm: INT;
END_VAR
SUPER^._InstancePath := THIS^.InstancePath; // Due to reflection its location is important

